# B&R Automation Studio project RS15_RX_30005_r00 (part 3)

#### A1_Basic.var - Local variables
```iecst
(********************************************************************
 * COPYRIGHT -- Microsoft
 ********************************************************************
 * Program: A1_Basic
 * File: A1_Basic.var
 * Author: pkiel
 * Created: July 11, 2011
 ********************************************************************
 * Local variables of program A1_Basic
 ********************************************************************)
VAR
	AutoAck : BOOL;
	AxisErrorNcAccess : UINT;
	DriveStatus : MC_DRIVESTATUS_TYP;
	HomeRestore : BOOL;
	InitEndlessPosition : BOOL;
	InitModPos_Done : BOOL;
	InitModPosition : BOOL;
  iiSetPosCount : DINT;
  iiSetPosCount1 : DINT;
  rSetPosCount1 : REAL;
  rMotorTemp : REAL;
  rAxisTimSet_SP_Vel  : REAL ; (*Set point Velocity for Axis manual timing setting cycle, in units/s*)
  rAxisTimSet_SP_Acc  : REAL ; (*Set point Acceleration for Axis manual timing setting cycle, in units/s²*)
  rAxisTimSet_SP_Dec  : REAL ; (*Set point Deceleration for Axis manual timing setting cycle, in units/s²*)
  uiAxisTimSet_SP_Dir : USINT ; (*Set point Direction for Axis manual timing setting cycle*)
  uiAxisTimSet_SP_ShiftAppMode : UINT ; (*Set point Shit Application mode for phasing Axis manual timing setting cycle*)
	MC_BR_InitEndlessPosition_0 : MC_BR_InitEndlessPosition;
	MC_BR_InitModPos_0 : MC_BR_InitModPos;
	MC_BR_Phasing_0 : MC_BR_Phasing;
	MC_BR_ReadDriveStatus_0 : MC_BR_ReadDriveStatus;
	MC_Home_0 : MC_Home;
	MC_Home_1 : MC_Home;
  MC_MoveVelocity_0 : MC_MoveVelocity;
  MC_MoveVelocity_1 : MC_MoveVelocity;
	MC_Power_0 : MC_Power;
	MC_ReadActualPosition_0 : MC_ReadActualPosition;
	MC_ReadActualTorque_0 : MC_ReadActualTorque;
	MC_ReadActualVelocity_0 : MC_ReadActualVelocity;
	MC_ReadAxisError_0 : MC_ReadAxisError;
	MC_ReadStatus_0 : MC_ReadStatus;
	MC_Reset_0 : MC_Reset;
  MC_Stop_0 : MC_Stop;
  MC_Stop_1 : MC_Stop;
  MC_SetOverride_0 : MC_SetOverride ;
	ResetError : BOOL;
  bTest_ : ARRAY[0..9] OF  BOOL;
  rTempActPhasDeg : REAL;
  rA9PosCorDeg : REAL;

  iiSP_SlPos_U  : DINT ; (*On Slave side, input set point position of the position controller ParID 428, in unit*)
  rSP_SlPos_Deg : REAL ; (*On Slave side, input set point position of the position controller ParID 428, in deg*)
  iiSP_MaPos_U  : DINT ; (*On Master side, input set point position of the position controller ParID 412, in unit*)
  rSP_MaPos_Deg : REAL ; (*On Master side, input set point position of the position controller ParID 412, in deg*)
  MC_BR_CyclicRead_0 : MC_BR_CyclicRead ;
  MC_BR_CyclicRead_1 : MC_BR_CyclicRead ;
  rTempPosA1_Deg : REAL;

  uiiMemoNumRev : UDINT ;
END_VAR
```

### Program Logical/BagMachine_Section/Perf/Axis1/A1_CamProfCalc

#### A1_CamProfCalc.var
```iecst
(********************************************************************
 * COPYRIGHT -- .
 ********************************************************************
 * Program: A1_CamProfCalc
 * File: A1_CamProfCalc.var
 * Author: dominique
 * Created: August 24, 2011
 ********************************************************************
 * Local variables of program A1_CamProfCalc
 ********************************************************************)

VAR
  stPerfCamSect : MC_CAM_SECTIONS_TYP ;
  stPerfCamProf : MC_CAMPROFILE_TYP ;
  MC_BR_CalcCamFromSections_0    : MC_BR_CalcCamFromSections ;
  MC_BR_DownloadCamProfileData_0 : MC_BR_DownloadCamProfileData ;
  MC_BR_GetCamMasterPosition_1   : MC_BR_GetCamMasterPosition ;
  MC_BR_GetCamMasterPosition_2   : MC_BR_GetCamMasterPosition ;
  MC_BR_GetCamSlavePosition_0    : MC_BR_GetCamSlavePosition ;
  MC_Home_0                      : MC_Home ;

  rMaInterval    : REAL ;
  rSlInterval    : REAL ;
  rSlPeriod      : REAL ;
  iiSlEndPoint   : DINT ;
  rSpeedInterval : REAL ;
  iStepCalPerfCam : INT ;
  bNextStep : BOOL ;
  bTestMode : BOOL ;

  iStepPosPerfCam : INT ;
  rCamMaPosition  : REAL ;
  rCamMaPos       : REAL ;
  rCamMaStartPos  : REAL ;
  rCamSlPosition  : REAL ;
  rCamSlPos       : REAL ;
  rCamSlPosCalc   : REAL ;
  rPosParkSlaveCamDeg   : REAL ;
  rTempPosParkSlaveCam  : REAL ;
  rTempPosParkMasterCam : REAL ;
  rMastMatchedSpeed : REAL ;
  bCmd_CalcCam_Test : BOOL ;
END_VAR

VAR CONSTANT

END_VAR
```

#### A1_CamProfCalcCyclic.st
```iecst
(********************************************************************
 * COPYRIGHT -- .
 ********************************************************************
 * Program: A1_CamProfCalc
 * File: A1_CamProfCalcCyclic.st
 * Author: dominique
 * Created: August 24, 2011
 ********************************************************************
 * Implementation of program A1_CamProfCalc
 ********************************************************************)

PROGRAM _CYCLIC

    IF ( gA[1].Cmd_CalcCameProf OR
         0                      OR
         bCmd_CalcCam_Test )    AND
       (iStepCalPerfCam = 0)    AND
       (iStepPosPerfCam = 0)    AND
       //0                        AND
       1                        THEN
      iStepCalPerfCam := 2 ;
    END_IF ;

    CASE iStepCalPerfCam OF

      // -------------------------------------------------------------------------------
      1 : ; // Waiting Error Reset
        IF EDGEPOS(gAlarmReset OR gA[1].Cmd_Reset) THEN
          g_bCamPerfCalcReset    := 0 ;
          g_bCamPerfCalc_Error   := 0 ;
          g_uiCalcCamPerfErrorID := 0 ;
          iStepCalPerfCam := 0 ;
        END_IF

      // -------------------------------------------------------------------------------
      2 : ; // Came profile calculation

        // Came profile calculation just for pos park on master side calculation
        // Synchro zone de 0° --> End Point of synchro zone
        // Compensation zone End Point of synchro zone --> Axis Periode

        // Calculation of Came section
        // Slave interval
        rSlInterval := gSP_A[1].MatchedSpeed * gA[1].UnitsPerDeg ;
        // Master interval
        rMaInterval := g_rActualSizePerf_in / gRecipeActive.Repeat * rSlInterval ;
        // Speed inteval
        rSpeedInterval := rSlInterval / rMaInterval ;
        // Slave Periode
        rSlPeriod := gA[1].AxisPeriod / gSP_PerfKnifeCount ;
        // Slave end point
        iiSlEndPoint := REAL_TO_DINT(rSlPeriod) ;
        // Master matched speed zone
        rMastMatchedSpeed := g_rActualSizePerf_in / gRecipeActive.Repeat * gSP_A[1].MatchedSpeed ;

        // First point of the Came Profile
        stPerfCamSect.Section[0].MasterPosition   := 0.0 ;
        stPerfCamSect.Section[0].SlavePosition    := 0.0 ;
        stPerfCamSect.Section[0].FirstDerivative  := rSpeedInterval ;
        stPerfCamSect.Section[0].SecondDerivative := 0.0 ;
        stPerfCamSect.Section[0].Mode             := mcABSOLUTE ;
        stPerfCamSect.Section[0].Type             := mcSTRAIGHT_LINE ;

        // Second point of the Came Profile
        stPerfCamSect.Section[1].MasterPosition   := rMaInterval ;
        stPerfCamSect.Section[1].SlavePosition    := rSlInterval ;
        stPerfCamSect.Section[1].FirstDerivative  := rSpeedInterval ;
        stPerfCamSect.Section[1].SecondDerivative := 0.0 ;
        stPerfCamSect.Section[1].Mode             := mcABSOLUTE ;
        stPerfCamSect.Section[1].Type             := mc5TH_ORDER_POLYNOMIAL ;

        // Third point of the Came Profile
        stPerfCamSect.Section[2].MasterPosition   := REAL_TO_DINT(gA[11].AxisPeriod) ;
        stPerfCamSect.Section[2].SlavePosition    := iiSlEndPoint ;
        stPerfCamSect.Section[2].FirstDerivative  := rSpeedInterval ;
        stPerfCamSect.Section[2].SecondDerivative := 0.0 ;
        stPerfCamSect.Section[2].Mode             := mcABSOLUTE ;
        stPerfCamSect.Section[2].Type             := mcLAST_POINT ;

        MC_BR_CalcCamFromSections_0.Execute           := 1 ;
        MC_BR_CalcCamFromSections_0.DataAddress       := ADR(stPerfCamSect) ;
        MC_BR_CalcCamFromSections_0.CamProfileAddress := ADR(stPerfCamProf) ;

        iStepCalPerfCam := 3 ;

      // -------------------------------------------------------------------------------
      3 : ; // Waiting result of the function
        IF MC_BR_CalcCamFromSections_0.Done AND
           ( bNextStep OR NOT(bTestMode) )  THEN
          MC_BR_CalcCamFromSections_0.Execute := 0 ;
          iStepCalPerfCam := 4 ;
          bNextStep := 0 ;
        ELSIF MC_BR_CalcCamFromSections_0.Error THEN
          g_uiCalcCamPerfErrorID := MC_BR_CalcCamFromSections_0.ErrorID;
          IF ( bNextStep OR NOT(bTestMode) ) THEN
            MC_BR_CalcCamFromSections_0.Execute :=0 ;
            g_bCamPerfCalc_Error := 1 ;
            bNextStep := 0 ;
            iStepCalPerfCam := 1 ;
          END_IF
        END_IF

      // -------------------------------------------------------------------------------
      4 : ; // Transfer Came to the Drive
        MC_BR_DownloadCamProfileData_0.Axis        := gA[1].Ident ;
        MC_BR_DownloadCamProfileData_0.DataAddress := ADR(stPerfCamProf) ;
        MC_BR_DownloadCamProfileData_0.Index       := g_uiIndexCamProfPerf ;
        MC_BR_DownloadCamProfileData_0.Periodic    := mcPERIODIC ;
        MC_BR_DownloadCamProfileData_0.Execute     := 1 ;

        iStepCalPerfCam := 5 ;

      // -------------------------------------------------------------------------------
      5 : ; // Waiting result of the function
        IF MC_BR_DownloadCamProfileData_0.Done AND
           ( bNextStep OR NOT(bTestMode) )     THEN
          MC_BR_DownloadCamProfileData_0.Execute:=FALSE;
          gA[1].Cmd_GetMaPosProf := 1 ;
          gA[1].Cmd_CalcCameProf := 0 ;
          bCmd_CalcCam_Test := 0 ;
          bNextStep := 0 ;
          iStepCalPerfCam := 0 ;
        ELSIF MC_BR_DownloadCamProfileData_0.Error THEN
          g_uiCalcCamPerfErrorID := MC_BR_DownloadCamProfileData_0.ErrorID;
          IF ( bNextStep OR NOT(bTestMode) ) THEN
            MC_BR_DownloadCamProfileData_0.Execute := 0 ;
            g_bCamPerfCalc_Error := 1 ;
            bNextStep := 0 ;
            iStepCalPerfCam := 1 ;
          END_IF
        END_IF
    END_CASE

    MC_BR_CalcCamFromSections_0() ;
    MC_BR_DownloadCamProfileData_0() ;

    // In Came Profile master position calculation according to the slave position
    IF ( gA[1].Cmd_GetMaPosProf   OR
         gA[1].Cmd_GetSlPosProf ) AND
       (iStepPosPerfCam = 0)      AND
       //0                          AND
       1                          THEN
      iStepPosPerfCam := 2 ;

      g_uiGetPosCamProfErrorID_1 := 0 ;
      g_uiGetPosCamProfErrorID_2 := 0 ;
      g_uiGetPosCamProfErrorID_3 := 0 ;
      g_uiHomCamProfErrorID      := 0 ;
    END_IF ;

    CASE iStepPosPerfCam OF
      // -------------------------------------------------------------------------------
      1 : ;// Waiting Error Reset
        IF EDGEPOS(gAlarmReset OR gA[1].Cmd_Reset) THEN
          iStepPosPerfCam := 0 ;
          g_bGetMaPosCamProfError_1 := 0 ;
          g_bGetMaPosCamProfError_2 := 0 ;
          g_bGetSlPosCamProfError   := 0 ;
          g_bHomeCamProfError       := 0 ;
        END_IF

      // -------------------------------------------------------------------------------
      2 : ; // Task selection
          IF gA[1].Cmd_GetMaPosProf THEN
            iStepPosPerfCam := 3 ;
          ELSIF gA[1].Cmd_GetSlPosProf THEN
            iStepPosPerfCam := 10 ;
          ELSE
            iStepPosPerfCam := 0 ;
          END_IF

      // -------------------------------------------------------------------------------
      3 : ; // Get Came master position command activation
        MC_BR_GetCamMasterPosition_1.Master := gA[11].Ident ;
        MC_BR_GetCamMasterPosition_1.Slave  := gA[1].Ident ;

        rCamSlPosCalc := H_FC_Modulus(IN_rMod:=rSlPeriod, IN_rVar:=gA[1].PositionCount) ;

        MC_BR_GetCamMasterPosition_1.Execute             := 1 ;
        MC_BR_GetCamMasterPosition_1.SlavePosition       := rCamSlPosCalc ;
        MC_BR_GetCamMasterPosition_1.MasterStartPosition := rCamMaStartPos ;
        MC_BR_GetCamMasterPosition_1.DataAddress         := ADR(stPerfCamProf) ;
        MC_BR_GetCamMasterPosition_1.MasterFactor        := 1 ;
        MC_BR_GetCamMasterPosition_1.SlaveFactor         := 1 ;
        IF MC_BR_GetCamMasterPosition_1.Done THEN
          rCamMaPosition := MC_BR_GetCamMasterPosition_1.MasterPosition ;
          MC_BR_GetCamMasterPosition_1.Execute := 0 ;
        ELSIF MC_BR_GetCamMasterPosition_1.Error THEN
          g_uiGetPosCamProfErrorID_1 := MC_BR_GetCamMasterPosition_1.ErrorID ;
          MC_BR_GetCamMasterPosition_1.Execute := 0 ;
          g_bGetMaPosCamProfError_1 := 1 ;
        END_IF

        MC_BR_GetCamMasterPosition_2.Master := gA[11].Ident ;
        MC_BR_GetCamMasterPosition_2.Slave  := gA[1].Ident ;

        rTempPosParkSlaveCam := gSP_A[1].ParkPosition * gA[1].UnitsPerDeg ;

        MC_BR_GetCamMasterPosition_2.Execute             := 1 ;
        MC_BR_GetCamMasterPosition_2.SlavePosition       := rTempPosParkSlaveCam ;
        MC_BR_GetCamMasterPosition_2.MasterStartPosition := rCamMaStartPos ;
        MC_BR_GetCamMasterPosition_2.DataAddress         := ADR(stPerfCamProf) ;
        MC_BR_GetCamMasterPosition_2.MasterFactor        := 1 ;
        MC_BR_GetCamMasterPosition_2.SlaveFactor         := 1 ;
        IF MC_BR_GetCamMasterPosition_2.Done AND
           NOT ( g_bGetMaPosCamProfError_1 ) THEN
          g_rPosParkMasterCam := MC_BR_GetCamMasterPosition_2.MasterPosition / gA[1].UnitsPerDeg ;
          MC_BR_GetCamMasterPosition_2.Execute := 0 ;
          iStepPosPerfCam := 4 ;
        ELSIF MC_BR_GetCamMasterPosition_2.Error THEN
          g_uiGetPosCamProfErrorID_2 := MC_BR_GetCamMasterPosition_2.ErrorID ;
          MC_BR_GetCamMasterPosition_2.Execute := 0 ;
          g_bGetMaPosCamProfError_2 := 1 ;
        END_IF

        IF g_bGetMaPosCamProfError_1 OR
           g_bGetMaPosCamProfError_2 THEN
          iStepPosPerfCam := 1 ;
        END_IF

      // -------------------------------------------------------------------------------
      4 : ; // Positionning Master on Synchro position
        MC_Home_0.Axis       := gA[11].Ident;
        IF gA[11].Ind_StandStill THEN
          MC_Home_0.Execute := 1 ;
        END_IF
        MC_Home_0.Position   := rCamMaPosition ;
        MC_Home_0.HomingMode := mcHOME_DIRECT;
        IF MC_Home_0.Done THEN
          MC_Home_0.Execute := 0 ;
          iStepPosPerfCam := 0 ;
          gA[1].Cmd_GetMaPosProf := 0 ;
          gA[1].Cmd_CalcCameProf := 0 ;
          g_bCameProf_OK := 1 ;
        ELSIF MC_Home_0.Error THEN
          g_uiHomCamProfErrorID := MC_Home_0.ErrorID ;
          MC_Home_0.Execute := 0 ;
          g_bHomeCamProfError := 1 ;
          iStepPosPerfCam := 1 ;
        END_IF

      // -------------------------------------------------------------------------------
      10 : ; // Get Came slave position command activation
        MC_BR_GetCamSlavePosition_0.Master := gA[11].Ident ;
        MC_BR_GetCamSlavePosition_0.Slave  := gA[1].Ident ;

        MC_BR_GetCamSlavePosition_0.Execute        := 1 ;
        MC_BR_GetCamSlavePosition_0.MasterPosition := rCamMaPos ;
        MC_BR_GetCamSlavePosition_0.DataAddress    := ADR(stPerfCamProf) ;
        MC_BR_GetCamSlavePosition_0.MasterFactor   := 1 ;
        MC_BR_GetCamSlavePosition_0.SlaveFactor    := 1 ;
        IF MC_BR_GetCamSlavePosition_0.Done THEN
          rCamSlPosition := MC_BR_GetCamSlavePosition_0.SlavePosition ;
          MC_BR_GetCamSlavePosition_0.Execute := 0 ;
          iStepPosPerfCam := 11 ;
        ELSIF MC_BR_GetCamSlavePosition_0.Error THEN
          g_uiGetPosCamProfErrorID_3 := MC_BR_GetCamSlavePosition_0.ErrorID ;
          MC_BR_GetCamSlavePosition_0.Execute := 0 ;
          g_bGetSlPosCamProfError := 1 ;
          iStepPosPerfCam := 1 ;
        END_IF

      // -------------------------------------------------------------------------------
      11 : ; //
        gA[1].Cmd_GetSlPosProf := 0 ;
        iStepPosPerfCam := 0 ;
      END_CASE

    MC_Home_0();
    MC_BR_GetCamMasterPosition_1() ;
    MC_BR_GetCamMasterPosition_2() ;
    MC_BR_GetCamSlavePosition_0() ;
END_PROGRAM
```

### Program Logical/BagMachine_Section/Perf/Axis1/A1_Control

#### A1_ControlCyclic.ld
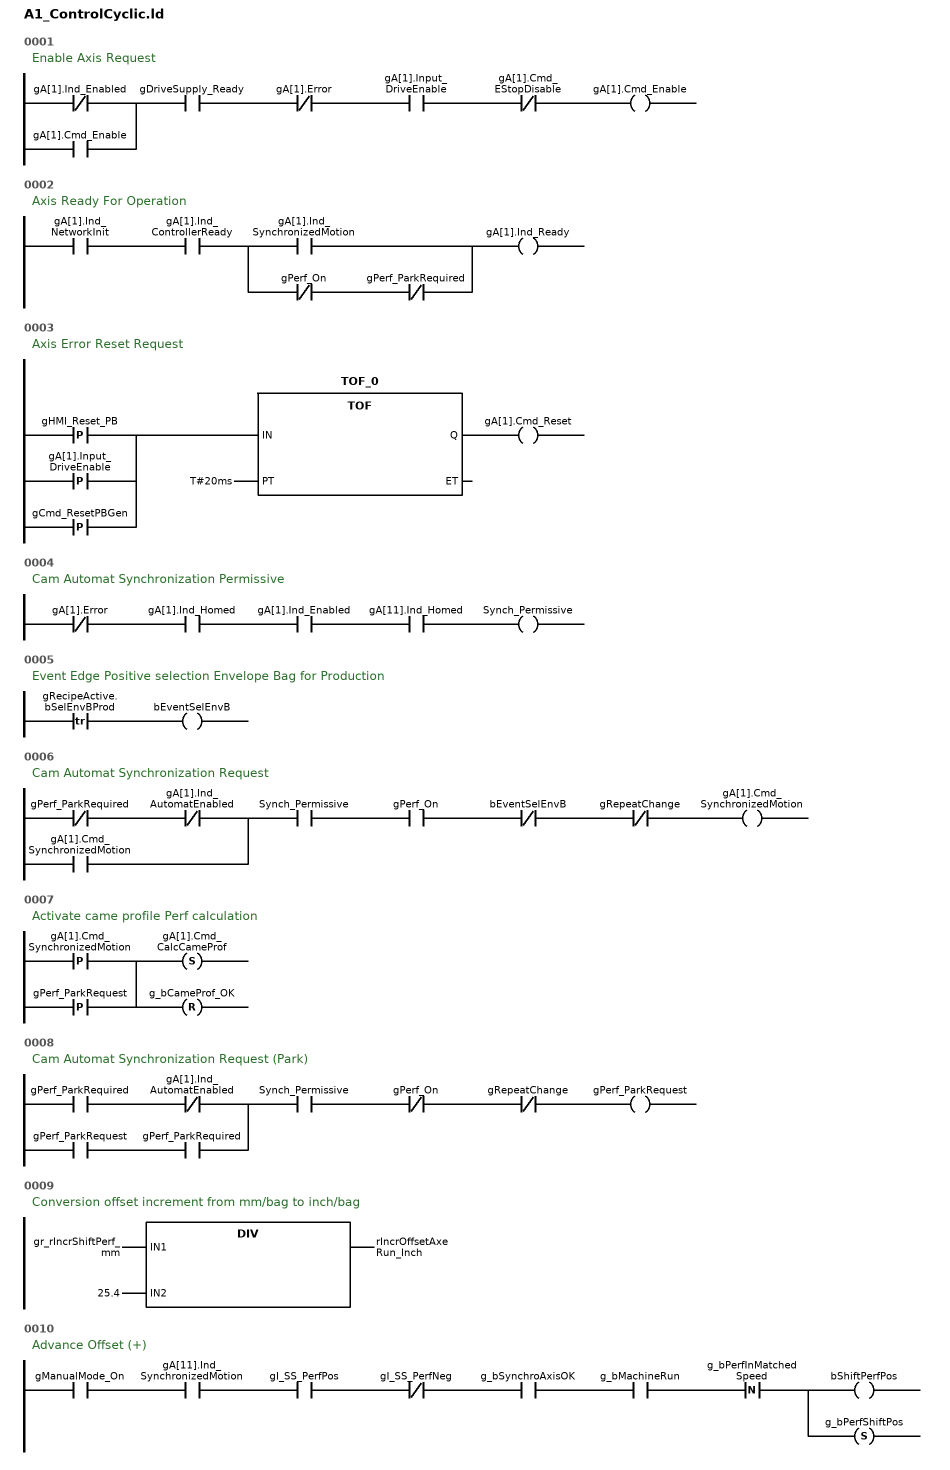
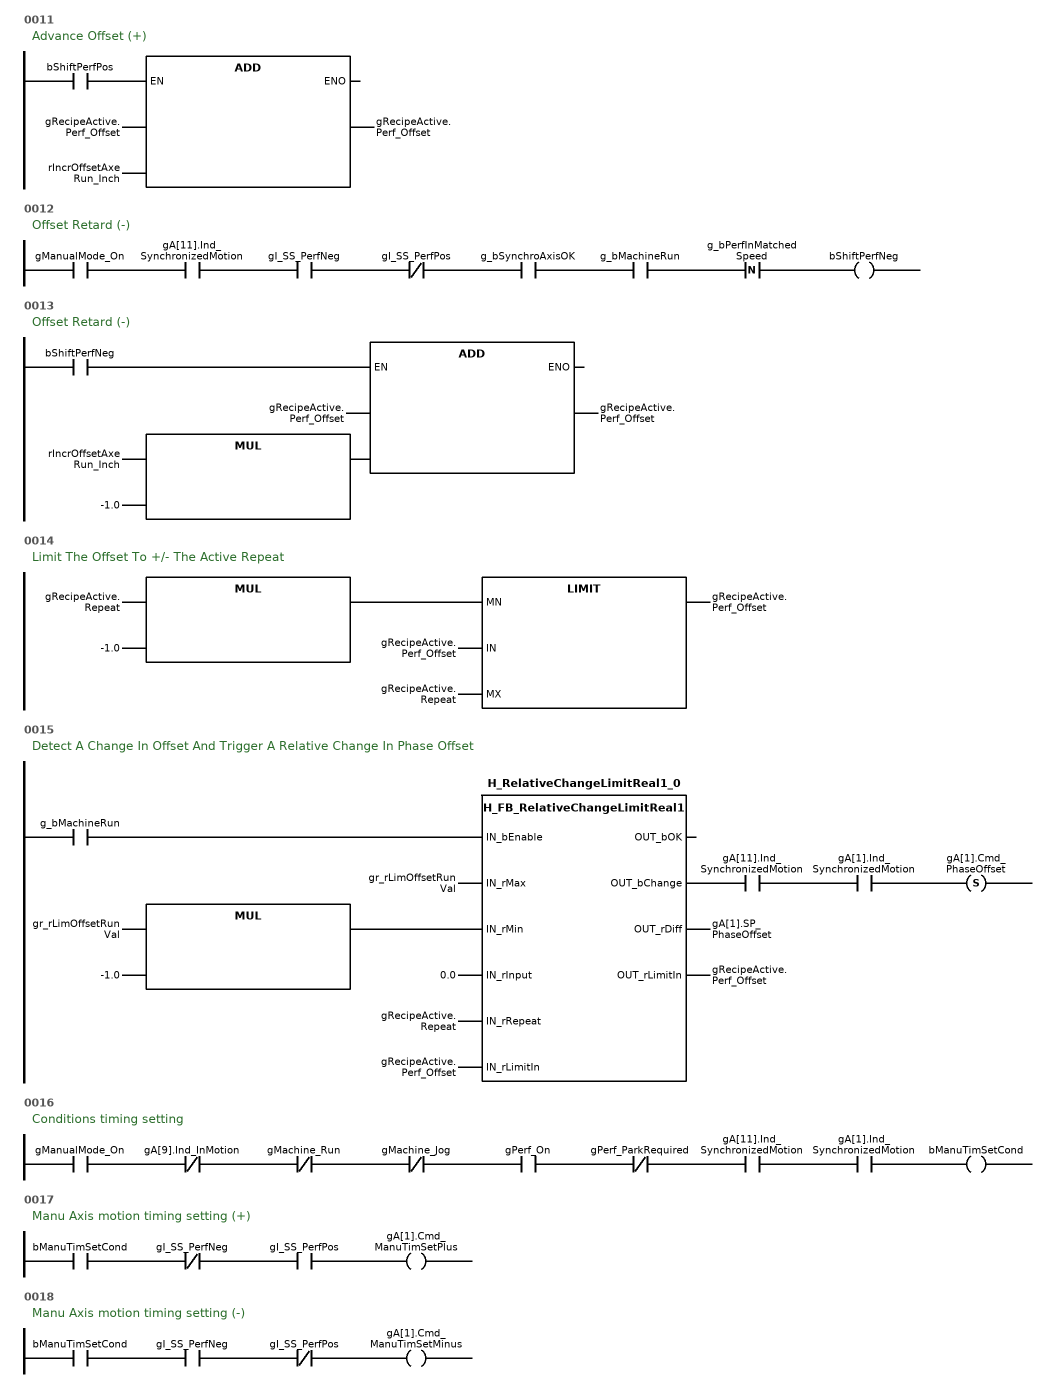
Ladder, written as Structured Text:
```iecst
(********************************************************************
 * COPYRIGHT -- Microsoft
 ********************************************************************
 * Program: A1_Control
 * File: A1_ControlCyclic.ld
 * Author: pkiel
 * Created: July 12, 2011
 ********************************************************************
 * Implementation of program A1_Control
 ********************************************************************)

PROGRAM _CYCLIC
VAR
    _p1 : BOOL;
    _e2 : R_TRIG;
    _e3 : R_TRIG;
    _e4 : R_TRIG;
    _e5 : R_TRIG;
    _e6 : R_TRIG;
    _e7 : F_TRIG;
    _p8 : BOOL;
    _e9 : F_TRIG;
END_VAR
(* Network 1: Enable Axis Request *)
gA[1].Cmd_Enable := (NOT gA[1].Ind_Enabled OR gA[1].Cmd_Enable) AND gDriveSupply_Ready AND NOT gA[1].Error AND gA[1].Input_DriveEnable AND NOT gA[1].Cmd_EStopDisable;

(* Network 2: Axis Ready For Operation *)
_p1 := gA[1].Ind_NetworkInit AND gA[1].Ind_ControllerReady;
gA[1].Ind_Ready := _p1 AND (gA[1].Ind_SynchronizedMotion OR (NOT gPerf_On AND NOT gPerf_ParkRequired));

(* Network 3: Axis Error Reset Request *)
_e2(CLK := gHMI_Reset_PB);
_e3(CLK := gA[1].Input_DriveEnable);
_e4(CLK := gCmd_ResetPBGen);
TOF_0(IN := _e2.Q OR _e3.Q OR _e4.Q, PT := T#20ms);
gA[1].Cmd_Reset := TOF_0.Q;

(* Network 4: Cam Automat Synchronization Permissive *)
Synch_Permissive := NOT gA[1].Error AND gA[1].Ind_Homed AND gA[1].Ind_Enabled AND gA[11].Ind_Homed;

(* Network 5: Event Edge Positive selection Envelope Bag for Production  *)
bEventSelEnvB := FALSE;

(* Network 6: Cam Automat Synchronization Request *)
gA[1].Cmd_SynchronizedMotion := ((NOT gPerf_ParkRequired AND NOT gA[1].Ind_AutomatEnabled) OR gA[1].Cmd_SynchronizedMotion) AND Synch_Permissive AND gPerf_On AND NOT bEventSelEnvB AND NOT gRepeatChange;

(* Network 7: Activate came profile Perf calculation  *)
_e5(CLK := gA[1].Cmd_SynchronizedMotion);
_e6(CLK := gPerf_ParkRequest);
IF _e5.Q OR _e6.Q THEN
    gA[1].Cmd_CalcCameProf := TRUE;
    g_bCameProf_OK := FALSE;
END_IF;

(* Network 8: Cam Automat Synchronization Request (Park) *)
gPerf_ParkRequest := ((gPerf_ParkRequired AND NOT gA[1].Ind_AutomatEnabled) OR (gPerf_ParkRequest AND gPerf_ParkRequired)) AND Synch_Permissive AND NOT gPerf_On AND NOT gRepeatChange;

(* Network 9: Conversion offset increment from mm/bag to inch/bag *)
rIncrOffsetAxeRun_Inch := gr_rIncrShiftPerf_mm / 25.4;

(* Network 10: Advance Offset (+) *)
_e7(CLK := g_bPerfInMatchedSpeed);
_p8 := gManualMode_On AND gA[11].Ind_SynchronizedMotion AND gI_SS_PerfPos AND NOT gI_SS_PerfNeg AND g_bSynchroAxisOK AND g_bMachineRun AND _e7.Q;
bShiftPerfPos := _p8;
IF _p8 THEN g_bPerfShiftPos := TRUE; END_IF;

(* Network 11: Advance Offset (+) *)
IF bShiftPerfPos THEN
    gRecipeActive.Perf_Offset := gRecipeActive.Perf_Offset + rIncrOffsetAxeRun_Inch;
END_IF;

(* Network 12: Offset Retard (-) *)
_e9(CLK := g_bPerfInMatchedSpeed);
bShiftPerfNeg := gManualMode_On AND gA[11].Ind_SynchronizedMotion AND gI_SS_PerfNeg AND NOT gI_SS_PerfPos AND g_bSynchroAxisOK AND g_bMachineRun AND _e9.Q;

(* Network 13: Offset Retard (-) *)
IF bShiftPerfNeg THEN
    gRecipeActive.Perf_Offset := gRecipeActive.Perf_Offset + (rIncrOffsetAxeRun_Inch * -1.0);
END_IF;

(* Network 14: Limit The Offset To +/- The Active Repeat *)
gRecipeActive.Perf_Offset := LIMIT(MN := gRecipeActive.Repeat * -1.0, IN := gRecipeActive.Perf_Offset, MX := gRecipeActive.Repeat);

(* Network 15: Detect A Change In Offset And Trigger A Relative Change In Phase Offset *)
H_RelativeChangeLimitReal1_0(IN_bEnable := g_bMachineRun, IN_rMax := gr_rLimOffsetRunVal, IN_rMin := gr_rLimOffsetRunVal * -1.0, IN_rInput := 0.0, IN_rRepeat := gRecipeActive.Repeat, IN_rLimitIn := gRecipeActive.Perf_Offset);
IF H_RelativeChangeLimitReal1_0.OUT_bChange AND gA[11].Ind_SynchronizedMotion AND gA[1].Ind_SynchronizedMotion THEN
    gA[1].Cmd_PhaseOffset := TRUE;
END_IF;
gA[1].SP_PhaseOffset := H_RelativeChangeLimitReal1_0.OUT_rDiff;
gRecipeActive.Perf_Offset := H_RelativeChangeLimitReal1_0.OUT_rLimitIn;

(* Network 16: Conditions timing setting  *)
bManuTimSetCond := gManualMode_On AND NOT gA[9].Ind_InMotion AND NOT gMachine_Run AND NOT gMachine_Jog AND gPerf_On AND NOT gPerf_ParkRequired AND gA[11].Ind_SynchronizedMotion AND gA[1].Ind_SynchronizedMotion;

(* Network 17: Manu Axis motion timing setting (+) *)
gA[1].Cmd_ManuTimSetPlus := bManuTimSetCond AND NOT gI_SS_PerfNeg AND gI_SS_PerfPos;

(* Network 18: Manu Axis motion timing setting (-) *)
gA[1].Cmd_ManuTimSetMinus := bManuTimSetCond AND gI_SS_PerfNeg AND NOT gI_SS_PerfPos;
END_PROGRAM
```

### Program Logical/BagMachine_Section/Perf/Axis1/A1_Cycle (IEC)

#### A1_CycleInit.st - Initialization code
```iecst
(********************************************************************
 * COPYRIGHT -- .
 ********************************************************************
 * Program: A1_Cycle
 * File: A1_CycleInit.st
 * Author: dominique
 * Created: August 01, 2011
 ********************************************************************
 * Implementation of program A1_Cycle
 ********************************************************************)

PROGRAM _INIT

(* TODO : Add your code here *)

END_PROGRAM
```

### A1_Init.ax
```
InitParameter (Version=2.24.0, NcSwId=ACP10)
  ACP10AXIS_typ:
    dig_in:
      level:
        reference = ncACTIV_HI
        pos_hw_end = ncACTIV_HI
        neg_hw_end = ncACTIV_HI
        trigger1 = ncACTIV_HI
        trigger2 = ncACTIV_HI
    encoder_if:
      parameter:
        count_dir = ncSTANDARD
        scaling:
          load:
            units = 18000
            rev_motor = 1
    limit:
      parameter:
        v_pos = 1.8e+006
        v_neg = 1.8e+006
        a1_pos = 5e+006
        a2_pos = 5e+006
        a1_neg = 5e+006
        a2_neg = 5e+006
        t_jolt = 0.0
        t_in_pos = 0.0
        pos_sw_end = 8388607
        neg_sw_end = -8388608
        ds_warning = 500.0
        ds_stop = 1000.0
        a_stop = 1e+030
        dv_stop = 0
        dv_stop_mode = ncOFF
    controller:
      mode = ncPOSITION
      position:
        kv = 400.0
        tn = 0.0
        t_predict = 0.0004
        t_total = 0.0012
        p_max = 1e+030
        i_max = 0.0
      speed:
        kv = 20.0
        tn = 0.0
        t_filter = 0.0
        isq_filter1:
          type = ncNOTCH
          a0 = 1321.0
          a1 = 400.0
          b0 = 0.0
          b1 = 0.0
          b2 = 0.0
          c0_par_id = 0
          c1_par_id = 0
        isq_filter2:
          type = ncOFF
          a0 = 0.0
          a1 = 0.0
          b0 = 0.0
          b1 = 0.0
          b2 = 0.0
          c0_par_id = 0
          c1_par_id = 0
        isq_filter3:
          type = ncOFF
          a0 = 0.0
          a1 = 0.0
          b0 = 0.0
          b1 = 0.0
          b2 = 0.0
          c0_par_id = 0
          c1_par_id = 0
      uf:
        type = ncLINEAR
        auto_config = ncMOTOR_PAR
        u0 = 0.0
        un = 0.0
        fn = 50.0
        k_f_slip = 0.0
      ff:
        torque_load = 0.0
        torque_pos = 0.0
        torque_neg = 0.0
        kv_torque = 0.0
        inertia = 0.0
        t_filter_a = 0.0
    move:
      stop:
        parameter[0]:
          decel_ramp = ncA_LIMIT
          controller = ncON
        parameter[1]:
          decel_ramp = ncA_LIMIT
          controller = ncON
        parameter[2]:
          decel_ramp = ncA_LIMIT
          controller = ncON
        parameter[3]:
          decel_ramp = ncA_LIMIT
          controller = ncON
        quickstop:
          decel_ramp = ncA_LIMIT
        drive_error:
          decel_ramp = ncA_LIMIT
      homing:
        parameter:
          s = 0
          v_switch = 5000.0
          v_trigger = 500.0
          a = 50000.0
          mode = ncHOME_OFFSET
          edge_sw = ncPOSITIVE
          start_dir = ncPOSITIVE
          trigg_dir = ncPOSITIVE
          ref_pulse = ncOFF
          tr_s_block = 0.0
      basis:
        parameter:
          v_pos = 36000.0
          v_neg = 100000.0
          a1_pos = 50000.0
          a2_pos = 50000.0
          a1_neg = 50000.0
          a2_neg = 50000.0
    message:
      text:
        parameter:
          format = ncBREAK
          columns = 80
          data_modul = Error_Eng
```

- Data object Logical/BagMachine_Section/Perf/Axis1/A1_Par (Apt) (no source held here)

### Program Logical/BagMachine_Section/Perf/Axis1/A1_Ref

#### A1_RefCyclic.ld
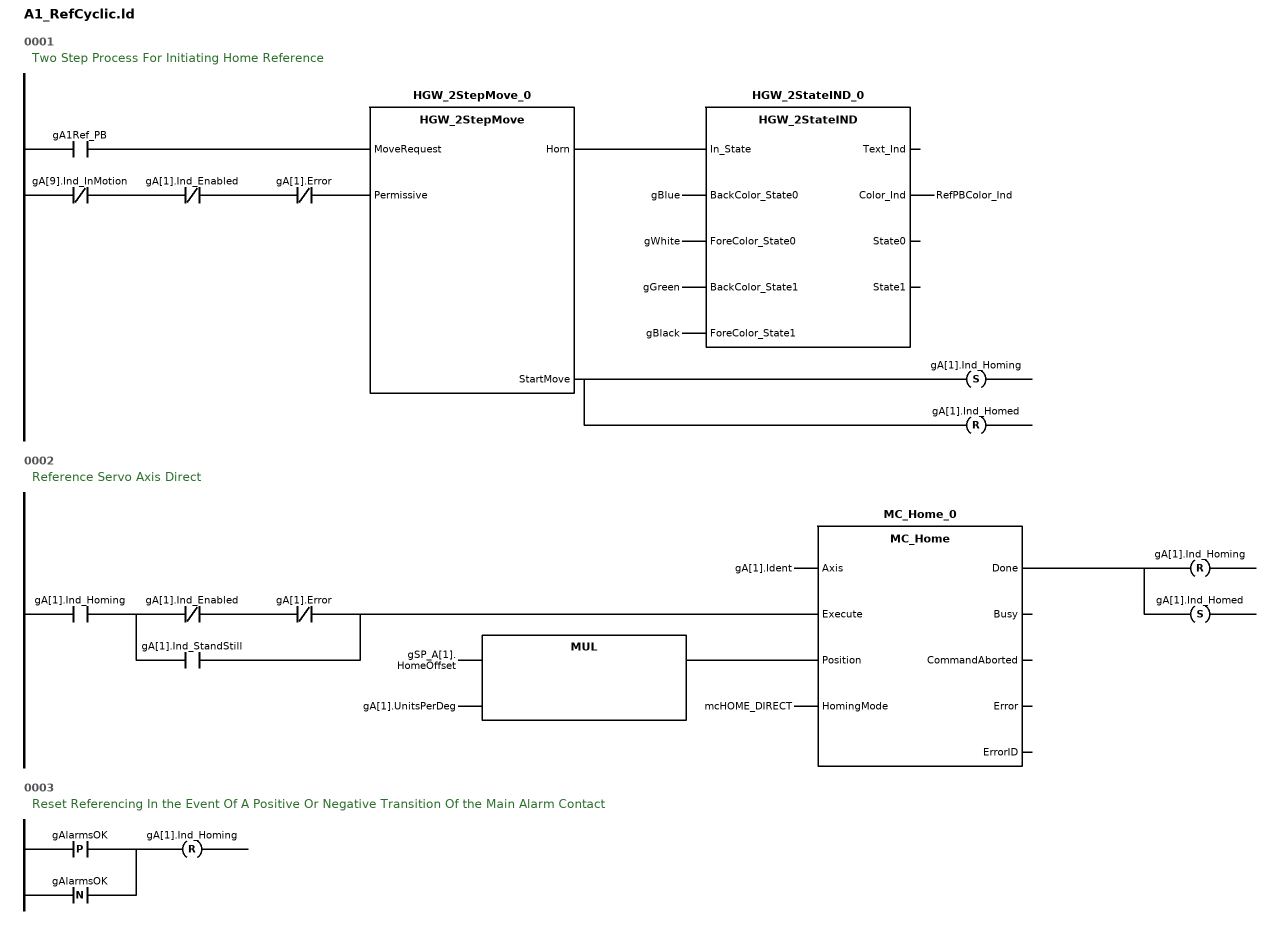
Ladder, written as Structured Text:
```iecst
(********************************************************************
 * COPYRIGHT -- Microsoft
 ********************************************************************
 * Program: A1_Ref
 * File: A1_RefCyclic.ld
 * Author: pkiel
 * Created: July 13, 2011
 ********************************************************************
 * Implementation of program A1_Ref
 ********************************************************************)

PROGRAM _CYCLIC
VAR
    _e1 : R_TRIG;
    _e2 : F_TRIG;
END_VAR
(* Network 1: Two Step Process For Initiating Home Reference *)
HGW_2StepMove_0(MoveRequest := gA1Ref_PB, Permissive := NOT gA[9].Ind_InMotion AND NOT gA[1].Ind_Enabled AND NOT gA[1].Error);
HGW_2StateIND_0(In_State := HGW_2StepMove_0.Horn, BackColor_State0 := gBlue, ForeColor_State0 := gWhite, BackColor_State1 := gGreen, ForeColor_State1 := gBlack);
RefPBColor_Ind := HGW_2StateIND_0.Color_Ind;
IF HGW_2StepMove_0.StartMove THEN
    gA[1].Ind_Homing := TRUE;
    gA[1].Ind_Homed := FALSE;
END_IF;

(* Network 2: Reference Servo Axis Direct *)
MC_Home_0(Axis := gA[1].Ident, Execute := gA[1].Ind_Homing AND ((NOT gA[1].Ind_Enabled AND NOT gA[1].Error) OR gA[1].Ind_StandStill), Position := gSP_A[1].HomeOffset * gA[1].UnitsPerDeg, HomingMode := mcHOME_DIRECT);
IF MC_Home_0.Done THEN
    gA[1].Ind_Homing := FALSE;
    gA[1].Ind_Homed := TRUE;
END_IF;

(* Network 3: Reset Referencing In the Event Of A Positive Or Negative Transition Of the Main Alarm Contact *)
_e1(CLK := gAlarmsOK);
_e2(CLK := gAlarmsOK);
IF _e1.Q OR _e2.Q THEN gA[1].Ind_Homing := FALSE; END_IF;
END_PROGRAM
```

- Data object Logical/BagMachine_Section/Perf/Axis11_VirtualAxis/A11_Init (Vax) - Virtual Axis Initialization File (no source held here)

- Data object Logical/BagMachine_Section/Perf/Axis11_VirtualAxis/A11_Par (Apt) - Virtual Axis Parameter File (no source held here)

### Program Logical/BagMachine_Section/Perf/Axis11_VirtualAxis/A11_Basic (IEC) - Basic Servo

#### A11_Basic.var
```iecst
(********************************************************************
 * COPYRIGHT -- Microsoft
 ********************************************************************
 * Program: A11_Basic
 * File: A11_Basic.var
 * Author: pkiel
 * Created: July 22, 2011
 ********************************************************************
 * Local variables of program A11_Basic
 ********************************************************************)
VAR
	AutoAck : BOOL;
	AxisErrorNcAccess : UINT;
	DriveStatus : MC_DRIVESTATUS_TYP;
	ErrorID : UINT;
	HomeRestore : BOOL;
	InitEndlessPosition : BOOL;
	InitModPos_Done : BOOL;
	InitModPosition : BOOL;
	MC_BR_InitEndlessPosition_0 : MC_BR_InitEndlessPosition;
	MC_BR_InitModPos_0 : MC_BR_InitModPos;
	MC_BR_Phasing_0 : MC_BR_Phasing;
  MC_BR_Phasing_1 : MC_BR_Phasing;
	MC_BR_ReadDriveStatus_0 : MC_BR_ReadDriveStatus;
	MC_Home_0 : MC_Home;
	MC_Home_1 : MC_Home;
	MC_MoveVelocity_0 : MC_MoveVelocity;
	MC_ReadActualPosition_0 : MC_ReadActualPosition;
	MC_ReadActualVelocity_0 : MC_ReadActualVelocity;
	MC_ReadAxisError_0 : MC_ReadAxisError;
	MC_ReadStatus_0 : MC_ReadStatus;
	MC_Reset_0 : MC_Reset;
	MC_Stop_0 : MC_Stop;
  stTON_O : TON ;
	ResetError : BOOL;
  rTemp_ : ARRAY[0..9] OF REAL ;
  bTest_ : ARRAY[0..9] OF BOOL ;
  rTest_ : ARRAY[0..9] OF REAL ;
  rAxisTimSet_SP_Vel  : REAL ; (*Set point Velocity for Axis manual timing setting cycle, in units/s*)
  rAxisTimSet_SP_Acc  : REAL ; (*Set point Acceleration for Axis manual timing setting cycle, in units/s²*)
  rAxisTimSet_SP_Dec  : REAL ; (*Set point Deceleration for Axis manual timing setting cycle, in units/s²*)
  uiAxisTimSet_SP_Dir : USINT ; (*Set point Direction for Axis manual timing setting cycle*)
  uiAxisTimSet_SP_ShiftAppMode : UINT ; (*Set point Shit Application mode for phasing Axis manual timing setting cycle*)
  rTempActPhasDeg : REAL;
  rA9PosCorDeg : REAL;
  MC_SetOverride_0 : MC_SetOverride;

  iiSP_SlPos_U  : DINT ; (*On Slave side, input set point position of the position controller ParID 428, in unit*)
  rSP_SlPos_Deg : REAL ; (*On Slave side, input set point position of the position controller ParID 428, in deg*)
  iiSP_MaPos_U  : DINT ; (*On Master side, input set point position of the position controller ParID 412, in unit*)
  rSP_MaPos_Deg : REAL ; (*On Master side, input set point position of the position controller ParID 412, in deg*)
  MC_BR_CyclicRead_0 : MC_BR_CyclicRead ;
  MC_BR_CyclicRead_1 : MC_BR_CyclicRead ;
  iIndex : INT;
  st_TON_0 : TON;
END_VAR
```

#### A11_BasicCyclic.st
```iecst
(********************************************************************
 * COPYRIGHT -- Microsoft
 ********************************************************************
 * Program: A11_Basic
 * File: A11_BasicCyclic.st
 * Author: pkiel
 * Created: July 22, 2011
 ********************************************************************
 * Implementation of program A11_Basic
 ********************************************************************)

PROGRAM _CYCLIC

	gA[11].UnitsPerInch := gA[11].AxisPeriod/gRecipeActive.Repeat;
  gA[11].InchPerDeg := gRecipeActive.Repeat / 360 ;

	IF (gA[11].Ident<>0) THEN

	(************************ READ DRIVE STATUS *************************)
	(* Access to the following bools:
	gA[x]_DriveStatus.Simulation			: If TRUE, simulation mode is active
	gA[x]_DriveStatus.NetworkInit			: If TRUE, the network is initialized
	gA[x]_DriveStatus.HomeSwitch			: If TRUE, the digital reference switch input is active
	gA[x]_DriveStatus.PosHWSwitch			: If TRUE, the positive hardware end switch is active
	gA[x]_DriveStatus.NegHWSwitch			: If TRUE, the negative hardware end switch is active
	gA[x]_DriveStatus.Trigger1				: If TRUE, the first trigger input is active
	gA[x]_DriveStatus.Trigger2				: If TRUE, the second trigger input is active
	gA[x]_DriveStatus.DriveEnable			: If TRUE, the enable input is active
	gA[x]_DriveStatus.ControllerReady		: If TRUE, the controller is ready to beturned on
	gA[x]_DriveStatus.ControllerStatus		: If TRUE, the controller is turned on (Same as MC_Power.Status)
	gA[x]_DriveStatus.AxisError				: If TRUE, at least one error has occurred (not acknowledged)
	gA[x]_DriveStatus.LagWarning			: If TRUE, the lag error has exceeded the limit value specified for a warning*)
		MC_BR_ReadDriveStatus_0.Enable := 1;
		MC_BR_ReadDriveStatus_0.Axis := gA[11].Ident;
		MC_BR_ReadDriveStatus_0.AdrDriveStatus := ADR (DriveStatus);
		MC_BR_ReadDriveStatus_0();
		gA[11].Ind_Simulation		:=	DriveStatus.Simulation;
		gA[11].Ind_NetworkInit		:=	DriveStatus.NetworkInit;
		gA[11].Input_Home			:=	DriveStatus.HomeSwitch;
		gA[11].Input_PosHW			:=	DriveStatus.PosHWSwitch;
		gA[11].Input_NegHW			:=	DriveStatus.NegHWSwitch;
		gA[11].Input_Trigger1		:=	DriveStatus.Trigger1;
		gA[11].Input_Trigger2		:=	DriveStatus.Trigger2;
		gA[11].Input_DriveEnable		:=	DriveStatus.DriveEnable;
		gA[11].Ind_ControllerReady	:=	DriveStatus.ControllerReady;
		gA[11].Ind_ControllerStatus	:=	DriveStatus.ControllerStatus;
		gA[11].Error					:=	DriveStatus.AxisError;
		gA[11].Ind_LagWarning		:=	DriveStatus.LagWarning;

	(************************ READ AXIS ERROR **********************)
		MC_ReadAxisError_0.Enable := gA[11].Ind_NetworkInit;
		MC_ReadAxisError_0.Axis := gA[11].Ident;
		MC_ReadAxisError_0.DataAddress := ADR(gA[11].ErrorText);
		MC_ReadAxisError_0.DataLength := SIZEOF(gA[11].ErrorText);
		MC_ReadAxisError_0.DataObjectName := 'Error_Eng';
		MC_ReadAxisError_0();
		IF(MC_ReadAxisError_0.Valid) THEN
			gA[11].ErrorID := MC_ReadAxisError_0.AxisErrorID;
			gA[11].ErrorCount := MC_ReadAxisError_0.AxisErrorCount;
		END_IF
	(* Auto Acknowledge Errors *)
		IF (gA[11].Cmd_Reset AND (gA[11].ErrorCount<>0) AND NOT AutoAck) THEN
			AutoAck:=1;
		ELSE
			AutoAck:=0;
		END_IF
	(*Axis Error Acknowledge*)
		IF (EDGEPOS(AutoAck) OR EDGEPOS(gA[11].ErrorAck)) THEN
			MC_ReadAxisError_0.Acknowledge := 1;
		ELSE;
			MC_ReadAxisError_0.Acknowledge :=0;
		END_IF

	(************************ RESET AXIS ERROR **********************)
		IF (gA[11].Cmd_Reset AND (gA[11].ErrorCount=0) AND gA[11].ErrorStop) THEN
			MC_Reset_0.Execute:=1;
		END_IF
		IF (MC_Reset_0.Done) THEN
			MC_Reset_0.Execute:=0;
			gA[11].Cmd_Reset:=0;
			ResetError := 0;
		END_IF
		IF (MC_Reset_0.Error) THEN
			MC_Reset_0.Execute:=0;
			gA[11].Cmd_Reset:=0;
			ResetError := 1;
		END_IF
		MC_Reset_0.Axis:=gA[11].Ident;
		MC_Reset_0();

	(************************ READ AXIS STATUS *************************)
		MC_ReadStatus_0.Enable := gA[11].Ind_NetworkInit;
		MC_ReadStatus_0.Axis := gA[11].Ident;
		MC_ReadStatus_0();
		IF(MC_ReadStatus_0.Valid = TRUE)THEN
			gA[11].Ind_Enabled 			:= NOT (MC_ReadStatus_0.Disabled);
			gA[11].Ind_StandStill		:= MC_ReadStatus_0.StandStill;
			gA[11].Ind_Stopping			:= MC_ReadStatus_0.Stopping;
			gA[11].Ind_DiscreteMotion	:= MC_ReadStatus_0.DiscreteMotion;
			gA[11].Ind_ContinuousMotion	:= MC_ReadStatus_0.ContinuousMotion;
			gA[11].Ind_SynchronizedMotion:= MC_ReadStatus_0.SynchronizedMotion;
			gA[11].ErrorStop				:= MC_ReadStatus_0.Errorstop;
		END_IF

	(******************** INIT POSITION MODULUS  *********************)
		MC_BR_InitModPos_0.Execute:= InitModPosition;
		MC_BR_InitModPos_0.Axis:= gA[11].Ident;
		MC_BR_InitModPos_0.Period:= REAL_TO_UDINT(gA[11].AxisPeriod);
		MC_BR_InitModPos_0.Factor:=1;
		InitModPos_Done:=MC_BR_InitModPos_0.Done;
		MC_BR_InitModPos_0();

	(******************** INIT ENDLESS POSITION *********************)
		MC_BR_InitEndlessPosition_0.Execute:= InitModPos_Done;
		MC_BR_InitEndlessPosition_0.Axis:= gA[11].Ident;
		MC_BR_InitEndlessPosition_0.DataAddress:= ADR(gEndPosData[11]);
		IF (MC_BR_InitEndlessPosition_0.Done) THEN
			InitModPosition:=0;
			InitEndlessPosition:=0;
			HomeRestore:=1;
		END_IF
		MC_BR_InitEndlessPosition_0();

	(************************ HOME AXIS FIRST POWER UP **********************)
		IF (HomeRestore AND NOT gA11_FirstHomed) THEN
			MC_Home_0.Execute:=1;
		END_IF
		MC_Home_0.Axis:=gA[11].Ident;
		MC_Home_0.Position:=0;
		MC_Home_0.HomingMode:=mcHOME_DIRECT;
		IF (MC_Home_0.Done) THEN
			MC_Home_0.Execute:=0;
			gA11_FirstHomed:=1;
		END_IF
		MC_Home_0();

	(************************ HOME AXIS **********************)
		IF (gA11_FirstHomed)     AND
       //NOT(gA[11].Ind_Homed) AND
       //g_bPerfInMatchedSpeed AND
       //gA[1].Ind_Homed       AND
       1                     THEN
			MC_Home_1.Execute:=HomeRestore;
		END_IF
		MC_Home_1.Axis:=gA[11].Ident;
		MC_Home_1.Position:=0;
		MC_Home_1.HomingMode:=mcHOME_RESTORE_POS;
		IF (MC_Home_1.Done) THEN
			gA[11].Ind_Homed:=1;
			HomeRestore:=0;
		END_IF
		MC_Home_1();

	(******************** READ ACTUAL POSITION *********************)
		MC_ReadActualPosition_0.Enable:= gA[11].Ind_NetworkInit;
		MC_ReadActualPosition_0.Axis:= gA[11].Ident;
		MC_ReadActualPosition_0();
		IF(MC_ReadActualPosition_0.Valid = TRUE)THEN
			gA[11].PositionCount := MC_ReadActualPosition_0.Position;
			gA[11].PositionInch := gA[11].PositionCount/gA[11].UnitsPerInch;
			gA[11].PositionDeg := gA[11].PositionCount/gA[11].UnitsPerDeg;
		END_IF

  //******************** READ SET POINT POSITION *********************
    // Slave side  : ParID 412 S_SET_VAX1 : 412: VAX: Position
    // Master side : ParID 412 S_SET_VAX1 : 412: VAX: Position

    // Slave side
    MC_BR_CyclicRead_0.Axis        := gA[11].Ident ;
    MC_BR_CyclicRead_0.Enable      := gA[11].Ind_NetworkInit;
    MC_BR_CyclicRead_0.ParID       := 412 ;
    MC_BR_CyclicRead_0.DataAddress := ADR(iiSP_SlPos_U);
    MC_BR_CyclicRead_0.DataType    := ncPAR_TYP_DINT ;
    // Master side
    MC_BR_CyclicRead_1.Axis        := gA[9].Ident ;
    MC_BR_CyclicRead_1.Enable      := gA[11].Ind_NetworkInit;
    MC_BR_CyclicRead_1.ParID       := 412 ;
    MC_BR_CyclicRead_1.DataAddress := ADR(iiSP_MaPos_U);
    MC_BR_CyclicRead_1.DataType    := ncPAR_TYP_DINT ;

    IF MC_BR_CyclicRead_0.Valid THEN
      rSP_SlPos_Deg := iiSP_SlPos_U/gA[11].UnitsPerDeg ;
    ELSIF MC_BR_CyclicRead_0.Error THEN
      MC_BR_CyclicRead_0.Enable := 0 ;
    END_IF
    IF MC_BR_CyclicRead_1.Valid THEN
      rSP_MaPos_Deg := iiSP_MaPos_U/gA[9].UnitsPerDeg ;
    ELSIF MC_BR_CyclicRead_1.Error THEN
      MC_BR_CyclicRead_1.Enable := 0 ;
    END_IF
    MC_BR_CyclicRead_0();
    MC_BR_CyclicRead_1();

  //******************** READ ACTUAL OFFSET *********************
  IF gA[11].rRSynDen > 0.0 THEN
    rTempActPhasDeg := rSP_SlPos_Deg - gA[11].rRSynNum / gA[11].rRSynDen * rSP_MaPos_Deg ;
    gA[11].rActPhasDeg := H_FC_Modulus (
                              IN_rMod := 360 * gA[11].rRSynNum / gA[11].rRSynDen ,
                              IN_rVar := rTempActPhasDeg
                                      ) ;
  END_IF

	(******************** READ ACTUAL VELOCITY *********************)
		IF(MC_ReadActualVelocity_0.Error=TRUE) THEN
			MC_ReadActualVelocity_0.Enable:= 0;
		ELSE
			MC_ReadActualVelocity_0.Enable:= 1;
		END_IF
		MC_ReadActualVelocity_0.Axis:= gA[11].Ident;
		MC_ReadActualVelocity_0();
		IF(MC_ReadActualVelocity_0.Valid = TRUE)THEN
			gA[11].ActualVelocity := MC_ReadActualVelocity_0.Velocity*60/gA[11].SP_MotorPPR;
			IF (gA[11].ActualVelocity>1) THEN
				gA[11].Ind_InMotion:=1;
			ELSE
				gA[11].Ind_InMotion:=0;
			END_IF
		END_IF

	(************************ AXIS VELOCITY MOVE **********************)
		MC_MoveVelocity_0.Axis:=gA[11].Ident;
		MC_MoveVelocity_0.Velocity:=gA[11].SP_Velocity*gA[11].AxisPeriod/60;
		MC_MoveVelocity_0.Acceleration:=gA[11].SP_Accel;
		MC_MoveVelocity_0.Deceleration:=gA[11].SP_Decel;
		MC_MoveVelocity_0.Direction:=mcPOSITIVE_DIR;
		IF ((EDGEPOS(gA[11].Cmd_ContinuousMotion)) OR (EDGEPOS(gA[11].Cmd_ContinuousMotionUpdate))) THEN
			MC_MoveVelocity_0.Execute:=1;
		ELSE
			MC_MoveVelocity_0.Execute:=0;
		END_IF;
		MC_MoveVelocity_0();

  //************************ AXIS OVERRIDE **********************
    MC_SetOverride_0.Axis      := gA[11].Ident ;
    MC_SetOverride_0.Enable    := gA[11].Cmd_Override ;
    MC_SetOverride_0.VelFactor := gA[11].rSP_OverrideV ;
    MC_SetOverride_0.AccFactor := gA[11].rSP_OverrideA ;
    IF (MC_SetOverride_0.Enabled) OR
       (MC_SetOverride_0.Error)   THEN
      gA[11].Cmd_Override := 0 ;
    END_IF
    MC_SetOverride_0();

	(************************ AXIS STOP **********************)
		MC_Stop_0.Axis:=gA[11].Ident;
		IF (gA[11].Ind_ContinuousMotion AND NOT gA[11].Cmd_ContinuousMotion) THEN
			MC_Stop_0.Deceleration:=gA[11].SP_Decel;
			MC_Stop_0.Execute:=1;
		END_IF
		IF (MC_Stop_0.Done OR MC_Stop_0.CommandAborted OR MC_Stop_0.Error) THEN
			MC_Stop_0.Execute:=0;
		END_IF
		MC_Stop_0();

    (************************ SHIFTING PERF CONTROL **********************)
    IF (g_iMachType = C_iRS26) THEN
      g_iNumBagPerfTear := REAL_TO_INT(gr_rDistPerfTearRS26_mm/gRecipeActive.Repeat/25.4) ;
      IF gA[12].bInMach THEN // Case Enveloppe Bag
        IF gRecipeActive.bSelEnvBProd THEN // Case Enveloppe Bag On
          g_iNumBagPerfTear := REAL_TO_INT(gr_rDistPerfTearEnvBOn_mm/gRecipeActive.Repeat/25.4) ;
        ELSE
          IF (g_rNumbPliers=2) THEN  // Case Enveloppe Bag Off and bags size 2 grippers
            g_iNumBagPerfTear := REAL_TO_INT(gr_rDistPerfTearEnvBOff2_mm/gRecipeActive.Repeat/25.4) ;
          ELSE                       // Case Enveloppe Bag Off and bags size 4 grippers
            g_iNumBagPerfTear := REAL_TO_INT(gr_rDistPerfTearEnvBOff4_mm/gRecipeActive.Repeat/25.4) ;
          END_IF
        END_IF
      END_IF
    ELSIF (g_iMachType = C_iRS15) THEN
      g_iNumBagPerfTear := REAL_TO_INT(gr_rDistPerfTearRS15_mm/gRecipeActive.Repeat/25.4) ;
    END_IF
    // Limit to avoid value out of array range
    g_iNumBagPerfTear := LIMIT(0,g_iNumBagPerfTear,C_iMaxBagPerfTear) ;

    IF gstCycA[1].CycManTimSet.CmdMov THEN
      g_iArrayBagPerfTear := g_iArrayBagPerfTearNul ;
      gA[1].Cmd_PhaseOffset := 0 ;
      g_iCountPerfShift[1] := 0 ;
      g_iCountPerfShift[2] := 0 ;
    END_IF;

    IF (g_iCountPerfShift[1] > 0)     AND
       EDGENEG(g_bPerfInMatchedSpeed) AND
       g_bMachineRun                  AND
       NOT(gRun_Stop)                 OR
       bTest_[1]                      THEN
       bTest_[1] := 0 ;
      FOR iIndex := g_iNumBagPerfTear-1 TO 1 BY -1 DO
        g_iArrayBagPerfTear[iIndex+1] := g_iArrayBagPerfTear[iIndex] ;
      END_FOR
      g_iArrayBagPerfTear[1] := 0 ;
    END_IF

    IF gA[1].Cmd_PhaseOffset THEN
      g_iCountPerfShift[1] := g_iCountPerfShift[1] + 1 ;
      g_iCountPerfShift[2] := g_iCountPerfShift[1] ;
      IF g_bPerfShiftPos THEN
        g_iArrayBagPerfTear[1] := 1 ;
      ELSE
        g_iArrayBagPerfTear[1] := -1 ;
      END_IF
      g_bPerfShiftPos := 0 ;
    END_IF

    (************************ AXIS PHASE CONTROL (Inches) **********************)
    MC_BR_Phasing_0.Slave:=gA[11].Ident;
    IF gA[1].Ind_SynchronizedMotion AND gA[11].Ind_SynchronizedMotion AND NOT(gstCycA[1].CycManTimSet.bSCyc) AND st_TON_0.Q THEN
      MC_BR_Phasing_0.Enable:=1;
    ELSE;
      MC_BR_Phasing_0.Enable:=0;
    END_IF;
    IF gA[1].Cmd_PhaseOffset  AND NOT(gstCycA[1].CycManTimSet.bSCyc) THEN
      MC_BR_Phasing_0.InitData:=1;
      gA[1].Cmd_PhaseOffset:=0;
      // Calculation new phase Drum/Master
      rTemp_[4] := gA[1].SP_PhaseOffset/gA[11].InchPerDeg ;
      rTemp_[5] := gRecipeActive.rPerf_PhasMasterDeg + rTemp_[4] ;
      gRecipeActive.rPerf_PhasMasterDeg := H_FC_Modulus (IN_rMod := 360, IN_rVar := rTemp_[5]) ;
      rTest_[0] := rTest_[0] + 1 ;
    ELSE
      MC_BR_Phasing_0.InitData:=0;
    END_IF
    MC_BR_Phasing_0.ApplicationMode     := mcMASTER_DISTANCE_BASED;
    MC_BR_Phasing_0.Shift               := gA[1].SP_PhaseOffset*gA[9].UnitsPerInch;
    MC_BR_Phasing_0.Velocity            := 6*gA[11].AxisPeriod/60;
    MC_BR_Phasing_0.Acceleration        := gA[11].SP_Decel;
    //MC_BR_Phasing_0.ApplicationDistance := 0.8*gA[9].AxisPeriod;
    MC_BR_Phasing_0.ApplicationDistance := 0.5*gA[9].AxisPeriod;
    MC_BR_Phasing_0.ShiftMode           := mcRELATIVE;
    MC_BR_Phasing_0();

    (************************ AXIS PHASE CONTROL (Inches) TIMING SETTING **********************)
    IF gstCycA[1].CycManTimSet.bSCyc THEN
      IF gA[1].Cmd_ManuTimSetPlus THEN
        rAxisTimSet_SP_Vel := gr_rAxisTimSet_SP_Vel*gA[9].AxisPeriod/60 / (gA[11].rRSynNum/gA[11].rRSynDen) ;
      ELSE
        rAxisTimSet_SP_Vel := - gr_rAxisTimSet_SP_Vel*gA[9].AxisPeriod/60 / (gA[11].rRSynNum/gA[11].rRSynDen) ;
      END_IF
        rAxisTimSet_SP_Acc := gr_rAxisTimSet_SP_Acc*gA[9].AxisPeriod/60/60 ;
    END_IF

    MC_BR_Phasing_1.Slave                  := gA[11].Ident;
    MC_BR_Phasing_1.Enable                 := gstCycA[1].CycManTimSet.bCyc ;
    MC_BR_Phasing_1.InitData               := gstCycA[1].CycManTimSet.bSCyc ;
    MC_BR_Phasing_1.PerformVelocityControl := gstCycA[1].CycManTimSet.CmdMov ;
    MC_BR_Phasing_1.Velocity               := rAxisTimSet_SP_Vel ;
    MC_BR_Phasing_1.Acceleration           := rAxisTimSet_SP_Acc ;
    MC_BR_Phasing_1.ApplicationMode        := mcVELOCITY_CONTROL ;
    MC_BR_Phasing_1();
    st_TON_0(IN:=NOT(MC_BR_Phasing_1.Enable),PT:=T#100ms) ;

    IF NOT(gstCycA[1].CycManTimSet.CmdMov) AND
       MC_BR_Phasing_1.ShiftAttained       OR
       NOT(gstCycA[1].CycManTimSet.bCyc)   OR
       MC_BR_Phasing_1.Error               AND
       1                                   THEN
      gstCycA[1].CycManTimSet.CmdStop := 0 ;
    END_IF
  END_IF
END_PROGRAM
```

#### A11_BasicInit.st
```iecst
(********************************************************************
 * COPYRIGHT -- Microsoft
 ********************************************************************
 * Program: A11_Basic
 * File: A11_BasicInit.st
 * Author: pkiel
 * Created: July 22, 2011
 ********************************************************************
 * Implementation of program A11_Basic
 ********************************************************************)

PROGRAM _INIT

	(* Axis Setpoint Variables *)
		gA[11].SP_MotorPPR := 36000;
		gA[11].SP_GearBoxInput:= 1;
		gA[11].SP_GearBoxOutput:= 1;
		gA[11].AxisPeriod := (gA[11].SP_MotorPPR*gA[11].SP_GearBoxInput/gA[11].SP_GearBoxOutput);
		gA[11].UnitsPerDeg := gA[11].AxisPeriod/360;
		gA[11].SP_Accel := 0.2*gA[11].AxisPeriod;
		gA[11].SP_Decel := 0.4*gA[11].AxisPeriod;
		gA[11].SP_EStopDecel := 3.0*gA[11].AxisPeriod;
		gA[11].SP_FStopDecel := 1.5*gA[11].AxisPeriod;
		gA[11].HomeVelocity:=12*gA[11].AxisPeriod/60.0;
    gA[11].rSP_CorPosVel := 0.0 ;
    gA[11].rSP_CorPosVel := 0.0 ;
    gA[11].rSP_OverrideV := 1.0 ;
    gA[11].rSP_OverrideA := 1.0 ;

    FOR iIndex := 0 TO C_iMaxBagPerfTear DO
      g_iArrayBagPerfTearNul[iIndex] := 0 ;
    END_FOR ;

	(* access master axis *)
		AxisErrorNcAccess := ncaccess(ncACP10MAN, ADR('Axis11'), ADR(gA[11].Ident));

	(* Trigger Initialization Of ModPosition *)
		InitModPosition:=1;

END_PROGRAM
```

- Program Logical/BagMachine_Section/Perf/Axis11_VirtualAxis/A11_Control (IEC) - Servo Control (no source held here)

### Program Logical/BagMachine_Section/Perf/Axis11_VirtualAxis/A11_Automat (IEC) - Cam Automat

#### A11_Automat.var - Local variables
```iecst
(********************************************************************
 * COPYRIGHT -- Microsoft
 ********************************************************************
 * Program: A11_Automat
 * File: A11_Automat.var
 * Author: pkiel
 * Created: July 22, 2011
 ********************************************************************
 * Local variables of program A11_Automat
 ********************************************************************)
VAR
  AutData : MC_AUTDATA_TYP;
  AutomatStart : BOOL;
  ErrorID : UINT;
  MasterParID : UINT;
  MC_BR_AutControl_0 : MC_BR_AutControl;
  MC_BR_InitMasterParIDTransfer_0 : MC_BR_InitMasterParIDTransfer;
  ParID_Ready : BOOL;
  PositionMOD : DINT;
  PositionOffset : DINT;
  SlaveStartOffset : REAL;
  Synch_Request : BOOL;
  usiMemoStat : USINT;
  InMatched : BOOL ;
  MatchedSpeed_Inch : REAL ;
  rTempPosA1_Inch   : REAL ;
  MasterOffset : REAL ;
  Value1 : DINT ;
  Value2 : DINT ;

END_VAR
```

### CamProfTest.cam
```
CamProfile (NcSwId=ACP10, MasterAxisVelocity=1, MasterAxisAcceleration=0, DefaultCurveType=Polynomial5, MathematicalNotation=true)
  FixPoint (x=360, IsMathX=true, y=180, IsDefinedDy=true, Dy=0.5, IsMathDy=true, IsDefinedDdy=false, Ddy=0, IsMathDdy=true, IsDefinedDddy=false, Dddy=0, IsMathDddy=true)
  Synchronline:
    LeftBoundary (IsFix=true, x=0, IsMathX=true, y=0)
    RightBoundary (IsFix=true, x=120, IsMathX=true, y=60)
    Gradient (Numerator=1, Denominator=2, IsMath=false, IsFix=false)
  Curve (Type=Polynomial5)
    LeftBoundary (IsDefinedDdy=false, Ddy=0, IsMathDdy=true, IsDefinedDddy=false, Dddy=0, IsMathDddy=true)
    RightBoundary (IsDefinedDdy=false, Ddy=0, IsMathDdy=true, IsDefinedDddy=false, Dddy=0, IsMathDddy=true)
    Spline3 (IsContinuous4Derivative=false, IsDefinedSaddlePoint=false, IsDefinedLineAs2ndSegment=false, IsDefinedSlopeOfLine=false, SlopeOfLine=0, IsMathSlopeOfLine=true)
    Supremum (y=1.7e+308, Dy=1.7e+308, IsMathDy=true, Ddy=1.7e+308, IsMathDdy=true, Dddy=1.7e+308, IsMathDddy=true)
    Infimum (y=-1.7e+308, Dy=-1.7e+308, IsMathDy=true, Ddy=-1.7e+308, IsMathDdy=true, Dddy=-1.7e+308, IsMathDddy=true)
  Cam (LeftBoundaryIndex=0, RightBoundaryIndex=1)
    Supremum (y=1.7e+308, Dy=1.7e+308, IsMathDy=true, Ddy=1.7e+308, IsMathDdy=true, Dddy=1.7e+308, IsMathDddy=true)
    Infimum (y=-1.7e+308, Dy=-1.7e+308, IsMathDy=true, Ddy=-1.7e+308, IsMathDdy=true, Dddy=1.7e+308, IsMathDddy=true)
  ChartExtensions
```

### Perf_Gen.typ
```iecst
(********************************************************************
 * COPYRIGHT -- Microsoft
 ********************************************************************
 * Program: Perf_Gen
 * File: Perf_Gen.typ
 * Author: pkiel
 * Created: July 19, 2011
 ********************************************************************
 * Local data types of program Perf_Gen
 ********************************************************************)

TYPE

  PerfPos : STRUCT

  END_STRUCT;

END_TYPE
```

### Perf_Gen.var
```iecst
(********************************************************************
 * COPYRIGHT -- Microsoft
 ********************************************************************
 * Program: Perf_Gen
 * File: Perf_Gen.var
 * Author: pkiel
 * Created: July 19, 2011
 ********************************************************************
 * Local variables of program Perf_Gen
 ********************************************************************)
VAR RETAIN
	HGW_2StatePB_0 : HGW_2StatePB;
END_VAR
VAR
	InParkPosition : BOOL;
	Perf_PB : BOOL;
	PerfColor_Ind : UINT;
	PerfText_Ind : UINT;
	RepeatMetric : INT;
	SecondKnife_Visibility : UINT;
	TON_0 : TON;
	rTempPosA1_Deg : REAL;
	rMatchSpeedPerf : REAL;
	H_FB_Flash_0 : H_FB_Flash;
  HMI_iEnvBPerfSetUpVisible : INT ;
  HMI_iPerfSetUpVisible : INT ;
END_VAR
```

### Package Logical/BagMachine_Section/FP - Axis

- Program Logical/BagMachine_Section/FP/FP_Gen (IEC) - General Flexo Press control (no source held here)

### Program Logical/BagMachine_Section/FP/FP_Dryer (IEC) - Dryer Control

#### DryerCyclic.st - Cyclic code
```iecst
(********************************************************************
 * COPYRIGHT -- .
 ********************************************************************
 * Program: FP_Dryer
 * File: FP_DryerCyclic.st
 * Author: dominique
 * Created: November 08, 2011
 ********************************************************************
 * Implementation of program FP_Dryer
 ********************************************************************)

PROGRAM _CYCLIC

    // -------------------------------------------------------------------
    // Temperature Sensor Alarme
    g_DRY_bTempSensorAlarm := (g_usiAI_DRY_Pt100_TempStatus = 3) ;

    // -------------------------------------------------------------------
    // Blower On/Off
    IF g_DRY_bBlowerAlarm           OR
       EDGENEG(gI_SS_MainPowerOff ) OR
       NOT(g_bMainPower_OnDelay)    OR
       g_bIndEStop                  THEN
      HMI_Cmd_BlowerOnPB := 0 ;
    END_IF ;

    IF HMI_Cmd_AutoOffDryOnPB THEN
      bQ_CR_DRY_Blower := HMI_Cmd_BlowerOnPB AND
                          g_bMachineRun      AND
                          1                  ;
    ELSE
      bQ_CR_DRY_Blower := HMI_Cmd_BlowerOnPB AND
                          1                  ;
    END_IF ;

    // Output activation
    gQ_CR_DRY_Blower := ( bQ_CR_DRY_Blower OR
                          stTOF_0.Q )      AND
                          NOT(g_bIndEStop) ;

    // HMI Blower PB Texte
    IF HMI_Cmd_BlowerOnPB THEN
      uiBlowerOnPBTxt_Ind := 1 ;
    ELSE
      uiBlowerOnPBTxt_Ind := 0 ;
    END_IF ;
    // HMI Dryer Auto Off PB Texte
    IF HMI_Cmd_AutoOffDryOnPB THEN
      uiAutoOffDryOnPBTxt_Ind := 7 ;
    ELSE
      uiAutoOffDryOnPBTxt_Ind := 6 ;
    END_IF ;

    // -------------------------------------------------------------------
    // Heater On/Off
    bActHeat := NOT(g_DRY_bHeaterAlarm) AND
                g_bMainPower_OnDelay    AND
                HMI_Cmd_BlowerOnPB      AND
                NOT(g_bIndEStop)        AND
                1                       ;

    g_DRY_bActHeat := gRecipeActive.bSelHeaterProd AND
                      bQ_CR_DRY_Blower             AND
                      bActHeat                     ;

    // Heater On delayed
    stTON_0(IN:=gQ_CR_DRY_HeatRegul,PT:=T#7s);
    bInd_NeedCool := stTON_0.Q      OR
                     g_DRY_bActHeat AND
                     stTOF_0.Q      ;

    // Blower Off delayed in oder to cool the Heater when switching Off Dryer
    stTOF_0(IN:=bInd_NeedCool,PT:=T#30s);
    rBlowerTimeRemain := (TIME_TO_REAL(stTOF_0.PT) - TIME_TO_REAL(stTOF_0.ET))/1000.0 ;
    // Blower Time Remaining Visible
    IF stTOF_0.Q             AND
       NOT(g_bMachineRun)    AND
       NOT(bQ_CR_DRY_Blower) THEN
      iTimRemVisible := 0 ;
    ELSE
      iTimRemVisible := 1 ;
    END_IF
    g_DRY_bIndCooling := stTOF_0.Q ;
    IF EDGENEG(gI_SS_MainPowerOff ) AND
       g_DRY_bIndCooling            THEN
      g_DRY_bMemPowerOff := 1 ;
    END_IF
    IF NOT(g_DRY_bIndCooling ) THEN
      g_DRY_bMemPowerOff := 0 ;
      g_DRY_bFlash := 0 ;
    END_IF
    H_FB_Flash_0(IN_bEnable:=g_DRY_bMemPowerOff, IN_rNumFlashPerSec:=2) ;
    g_DRY_bFlash := H_FB_Flash_0.OUT_bFlash ;

    // HMI Heater PB Texte
    IF gRecipeActive.bSelHeaterProd THEN
      uiHeaterOnPBTxt_Ind := 3 ;
    ELSE
      uiHeaterOnPBTxt_Ind := 2 ;
    END_IF ;

    // Dryer activated
    g_bSelDryerProd := gRecipeActive.bSelHeaterProd OR
                       HMI_Cmd_BlowerOnPB           OR
                       bTest                        ;

END_PROGRAM
```

### Program Logical/BagMachine_Section/FP/FP_Heater (IEC) - A new program

#### FP_HeaterCyclic.st - Cyclic code
```iecst
(********************************************************************
 * COPYRIGHT -- .
 ********************************************************************
 * Program: FP_Heater
 * File: FP_HeaterCyclic.st
 * Author: dominique
 * Created: August 22, 2012
 ********************************************************************
 * Implementation of program FP_Heater
 ********************************************************************)

PROGRAM _CYCLIC

//------------------------------------------------------------------
// Lecture sonde de temperature
  rSondeTempRegTDegC[1] := INT_TO_REAL(gAI_DRY_Pt100_Temp) / 10.0 ;
  rSondeTempRegTDegF[1] := rSondeTempRegTDegC[1] * 9/5 + 32 ;

  // -------------------------------------------------------------------
  // Temperature Sensor Alarme
  g_DRY_bTempSensorAlarm := (g_usiAI_DRY_Pt100_TempStatus = 3) ;

  // Limit operator Setpoint
  gRecipeActive.rHeatSPDegF := LIMIT(rBornInfConsTempChauf[1],gRecipeActive.rHeatSPDegF,rBornSupConsTempChauf[1]) ;

  // Parametre mesure de temperature du regulateur
  IF g_DRY_bActHeat AND NOT(g_DRY_bTempSensorAlarm) AND NOT(g_bIndEStop) THEN
    rMesTempRegTChauf[1] := rSondeTempRegTDegF[1] ;
  ELSE
    rMesTempRegTChauf[1] := gRecipeActive.rHeatSPDegF ;
  END_IF;

  // Calcul periode echantillonnage appel PID, en s
  // TSI#cycleTime : Temps de cyle de la tache cyclique d appel du regulateur, en ms ( normalmement = 30ms )
  iiRegTChauf_TC[1] := 20 ;
  // Periode appel boucle PID
  rRegTChauf_T[1] := 2 ;

  // Valeur filtree de l'erreur
  // Y = 1/(1+t/T)E + 1/(1+T/t)Y_1
  IF ( rRegTChauf_T[1] <> 0 ) AND
     ( rPT1_t <> 0 )          THEN
    rRegTChauf_ErrF_1[1] := rRegTChauf_ErrF[1] ;
    rRegTChauf_ErrF[1] := ( 1/(1+rPT1_t/rRegTChauf_T[1]) * rRegTChauf_Err[1] + 1/(1+rRegTChauf_T[1]/rPT1_t) * rRegTChauf_ErrF_1[1] ) ;
  END_IF;

  // Appel du PID tout les n cycles PWM
  IF iCptSeuilAppelRegTChauf[1] >= iSeuilAppelPID_RegTChauf[1] THEN
    // Calcul nouvelle erreur
    rRegTChauf_Err[1] := ( gRecipeActive.rHeatSPDegF - rMesTempRegTChauf[1] ) ;
    // Calcul terme proportionnel
    rRegTChauf_TP[1] := rPIDRegTChaufKP[1] * rRegTChauf_Err[1] ;
    // Calcul terme Integral
    IF rPIDRegTChaufKI[1] <> 0.0 THEN  // Traitement cas division par 0
      rRegTChauf_TI[1] := rRegTChauf_TI_1[1] + rRegTChauf_T[1] * 1/rPIDRegTChaufKI[1] * rRegTChauf_Err[1] ;
    ELSE
      rRegTChauf_TI[1] := 0 ;
    END_IF;
    // Init terme Integral sur desactivation regul
    IF g_bIndEStop OR rRegTChauf_TI[1] < 0 OR rRegTChauf_TI_1[1] < 0 OR g_DRY_bTempSensorAlarm THEN
      rRegTChauf_TI[1]   := 0 ;
      rRegTChauf_TI_1[1] := 0 ;
    END_IF;
    // Limitation val sup terme Integral lorsque sortie saturee
    IF rRegTChauf_YPC[1] >= 100 THEN
      rRegTChauf_TI[1] := rRegTChauf_TI_1[1] ;
    END_IF;
    rRegTChauf_TI_1[1] := rRegTChauf_TI[1] ;
    // Calcul terme Derive
    IF rRegTChauf_T[1] <> 0.0 THEN  // Traitement cas division par 0
      rDiff_ErrF[1] := ( rRegTChauf_ErrF[1] - rRegTChauf_Err_1[1] ) ;
      rRegTChauf_TD[1] := 1/rRegTChauf_T[1] * rPIDRegTChaufKD[1] * rDiff_ErrF[1] ;
      // Memo erreur filtree
      rRegTChauf_Err_1[1] := rRegTChauf_ErrF[1] ;
    ELSE
      rRegTChauf_TD[1] := 0 ;
    END_IF;
    // Calcul sortie
    rRegTChauf_Y[1] := rRegTChauf_TP[1] + rRegTChauf_TI[1] + rRegTChauf_TD[1] ;
    // Conversion sortie en %
    IF rBornSupConsTempChauf[1] <> 0.0 THEN  // Traitement cas division par 0
      rRegTChauf_YPC[1] := rRegTChauf_Y[1] /rBornSupConsTempChauf[1] * 100 ;
    ELSE
      rRegTChauf_YPC[1] := 0 ;
    END_IF;
    IF rRegTChauf_YPC[1] > 100 THEN
      rRegTChauf_YPC[1] := 100 ;
    END_IF;
    IF rRegTChauf_YPC[1] < 0 OR g_DRY_bTempSensorAlarm OR g_bIndEStop OR NOT(g_DRY_bActHeat) THEN
      rRegTChauf_YPC[1] := 0 ;
    END_IF;
  END_IF;

  // Appel bloc PID
  // Incrementation et remise a zero du compteur d'appel du PID
  iSeuilAppelPID_RegTChauf[1] := 100 ; // Pour une tache interruptive de 20ms 100x20 = 2000ms = 2s
  iCptSeuilAppelRegTChauf[1]  := iCptSeuilAppelRegTChauf[1]  + 1  ;
  IF iCptSeuilAppelRegTChauf[1] > iSeuilAppelPID_RegTChauf[1] THEN
    iCptSeuilAppelRegTChauf[1] := 0 ;
  END_IF;

  // Parametres du PWM
  LCRPWM_0[1].enable      := 1 ;
  LCRPWM_0[1].x           := rRegTChauf_YPC[1] ;
  LCRPWM_0[1].max_value   := 100.0 ;
  LCRPWM_0[1].min_value   := 0.0 ;
  LCRPWM_0[1].t_min_pulse := iiRegTChauf_TC[1] / 1000 ;
  LCRPWM_0[1].t_period    := rRegTChauf_T[1] ;
  LCRPWM_0[1]() ;

  // Activation de la sortie regulee
  IF g_DRY_bActHeat AND NOT(g_DRY_bTempSensorAlarm) AND NOT(g_bIndEStop) THEN
    bImdoRT_ActChauf[1] := LCRPWM_0[1].pulse AND NOT(bTest) ;
  ELSE
    bImdoRT_ActChauf[1] := 0 ;
  END_IF;
  gQ_CR_DRY_HeatRegul := bImdoRT_ActChauf[1] ;

  // Calcul pic de chauffe a l'activation du chauffage
  IF EDGEPOS(g_DRY_bActHeat) THEN
    bImpulsDemarSech := 1 ;
  END_IF ;
  IF rSondeTempRegTDegF[1] >= gRecipeActive.rHeatSPDegF - rDeltaTStopPicChauf THEN
    bImpulsDemarSech := 0 ;
  END_IF ;

  // Batterie de chauffe TOR
  IF gRecipeActive.rHeatSPDegF > rSeuilConsTempActBattTOR OR
    bImpulsDemarSech                                      THEN
    gQ_CR_DRY_HeatContinu := g_DRY_bActHeat AND NOT(bTest);
  ELSE
    gQ_CR_DRY_HeatContinu := 0 ;
  END_IF ;

  // Conversion for trending
  IF ( gInchMetric_Ind = 2 ) THEN
    rTrendActTempRegT[1]   := rSondeTempRegTDegC[1] ;
    rTrendSetPTempRegT[1]  := (gRecipeActive.rHeatSPDegF-32) * 5/9 ;
    rTrendRegTChauf_Err[1] := (rRegTChauf_Err[1]-32) * 5/9 ;
  ELSE
    rTrendActTempRegT[1]   := rSondeTempRegTDegF[1] ;
    rTrendSetPTempRegT[1]  := gRecipeActive.rHeatSPDegF ;
    rTrendRegTChauf_Err[1] := rRegTChauf_Err[1] ;
  END_IF;

END_PROGRAM
```

- Data object Logical/BagMachine_Section/FP/Axis2/A2_Init (Ax) - Servo Axis Initialization File (no source held here)

### Data object Logical/BagMachine_Section/FP/Axis2/A2_Par (Apt) - Servo Axis Parameter File

#### A2_Par.apt
```
AcoposParameterTable:
  Root Parameters:
    110 = ncSW_OFF (Name=CMD_SIMULATION)  // Simulation mode: Command
    128 = 1 (Name=SGEN_SW_END_IGNORE)  // SGEN_SW_END_IGNORE
    Axis Parameter Identification Induction Motor:
      General Parameters:
        30 = 1 (Name=MOTOR_TYPE)  // Motor: Type
        31 = 515 (Name=MOTOR_COMPATIBILITY)  // Motor: Software compatibility
        46 = 1 (Name=MOTOR_WIND_CONNECT)  // Motor: Winding connection
        62 = 0.109 (Name=MOTOR_INERTIA, Unit=kgm²)  // Motor: Moment of inertia
        849 = 0 (Name=MOTOR_TAU_THERM, Unit=s)  // Motor: Thermal time constant
      Brake Parameters:
        42 = 0 (Name=MOTOR_BRAKE_CURR_RATED, Unit=A)  // Motor holding brake: Rated current
        43 = 0 (Name=MOTOR_BRAKE_TORQ_RATED, Unit=Nm)  // Motor holding brake: Rated torque
        44 = 0 (Name=MOTOR_BRAKE_ON_TIME, Unit=s)  // Motor holding brake: Engaging delay
        45 = 0 (Name=MOTOR_BRAKE_OFF_TIME, Unit=s)  // Motor holding brake: Release delay
      Thermo Sensor Parameters:
        64 = 391 (Name=MOTOR_TEMPSENS_PAR1)  // Temperature sensor: Parameter 1
        65 = 1492 (Name=MOTOR_TEMPSENS_PAR2)  // Temperature sensor: Parameter 2
        66 = -30 (Name=MOTOR_TEMPSENS_PAR3)  // Temperature sensor: Parameter 3
        67 = 12.01 (Name=MOTOR_TEMPSENS_PAR4)  // Temperature sensor: Parameter 4
        68 = 45.98 (Name=MOTOR_TEMPSENS_PAR5)  // Temperature sensor: Parameter 5
        69 = 75.71 (Name=MOTOR_TEMPSENS_PAR6)  // Temperature sensor: Parameter 6
        70 = 102.2 (Name=MOTOR_TEMPSENS_PAR7)  // Temperature sensor: Parameter 7
        71 = 126.41 (Name=MOTOR_TEMPSENS_PAR8)  // Temperature sensor: Parameter 8
        72 = 148.88 (Name=MOTOR_TEMPSENS_PAR9)  // Temperature sensor: Parameter 9
        73 = 170 (Name=MOTOR_TEMPSENS_PAR10)  // Temperature sensor: Parameter 10
        74 = 100 (Name=MOTOR_WIND_TEMP_MAX, Unit=°C)  // Temperature sensor: Limit temperature
      Result Parameters of Parameter Identification:
        47 = 2 (Name=MOTOR_POLEPAIRS)  // Motor: Number of pole-pairs
        48 = 322 (Name=MOTOR_VOLTAGE_RATED, Unit=V)  // Motor: Rated voltage
        49 = 0 (Name=MOTOR_VOLTAGE_CONST, Unit=mV*min)  // Motor: Voltage constant
        50 = 1000 (Name=MOTOR_SPEED_RATED, Unit=1/min)  // Motor: Rated speed
        51 = 8000 (Name=MOTOR_SPEED_MAX, Unit=1/min)  // Motor: Maximum speed
        52 = 162.34 (Name=MOTOR_TORQ_STALL, Unit=Nm)  // Motor: Stall torque
        53 = 162.34 (Name=MOTOR_TORQ_RATED, Unit=Nm)  // Motor: Rated torque
        54 = 577.34 (Name=MOTOR_TORQ_MAX, Unit=Nm)  // Motor: Peak torque
        55 = 0 (Name=MOTOR_TORQ_CONST, Unit=Nm/A)  // Motor: Torque constant
        56 = 40.69 (Name=MOTOR_CURR_STALL, Unit=A)  // Motor: Stall current
        57 = 40.69 (Name=MOTOR_CURR_RATED, Unit=A)  // Motor: Rated current
        58 = 238.47 (Name=MOTOR_CURR_MAX, Unit=A)  // Motor: Peak current
        59 = 0 (Name=MOTOR_WIND_CROSS_SECT, Unit=mm²)  // Motor: Line cross section
        60 = 0.1542 (Name=MOTOR_STATOR_RESISTANCE, Unit=Ohm)  // Motor: Stator resistance
        61 = 0.00180 (Name=MOTOR_STATOR_INDUCTANCE, Unit=Henry)  // Motor: Stator inductance
        63 = 0 (Name=MOTOR_COMMUT_OFFSET, Unit=rad)  // Motor: Commutation offset
        76 = 0.10915 (Name=MOTOR_ROTOR_RESISTANCE, Unit=Ohm)  // Motor: Rotor resistance
        77 = 0.00180 (Name=MOTOR_ROTOR_INDUCTANCE, Unit=Henry)  // Motor: Rotor inductance
        78 = 0.0527 (Name=MOTOR_MUTUAL_INDUCTANCE, Unit=Henry)  // Motor: Mutual inductance
        79 = 18.5 (Name=MOTOR_MAGNETIZING_CURR, Unit=A)  // Motor: Magnetizing current
```

### Program Logical/BagMachine_Section/FP/Axis2/A2_Control (IEC) - Servo Control

#### A2_Control.var
```iecst
(********************************************************************
 * COPYRIGHT -- Microsoft
 ********************************************************************
 * Program: A2_Control
 * File: A2_Control.var
 * Author: Dominique
 * Created: October 15, 2011
 ********************************************************************
 * Local variables of program A2_Control
 ********************************************************************)
VAR
	HGW_ChangeReal_0 : HGW_ChangeReal;
	HGW_RelativeChangeReal_0 : H_FB_RelativeChangeLimitReal1;
	HGW_Toggle_0 : HGW_Toggle;
	Synch_Permissive : BOOL;
	TOF_0 : TOF;
	TON_0 : TON;
  rIncrOffsetAxeRun_Inch : REAL ;
  rPoub : ARRAY[0..5] OF REAL ;
  bCmd_ManuTimSet : BOOL ;

  HMI_Cmd_ManuTimSetPlus : BOOL ;
  bLockSP_OffsetPrintRol : BOOL ;
END_VAR
```

#### A2_ControlCyclic.ld
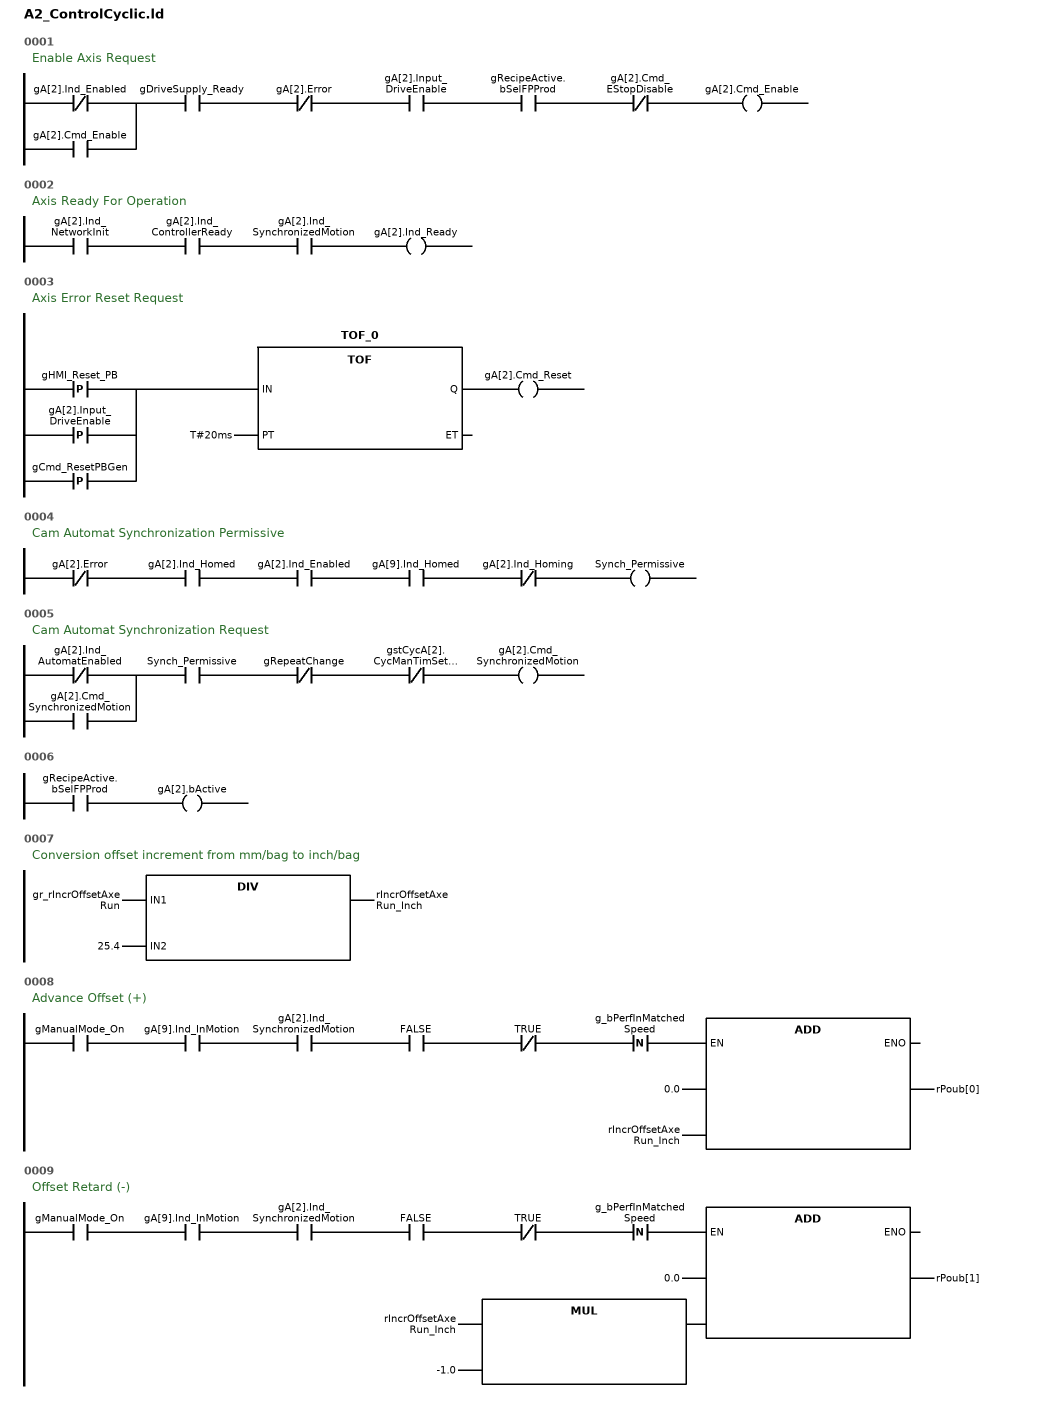
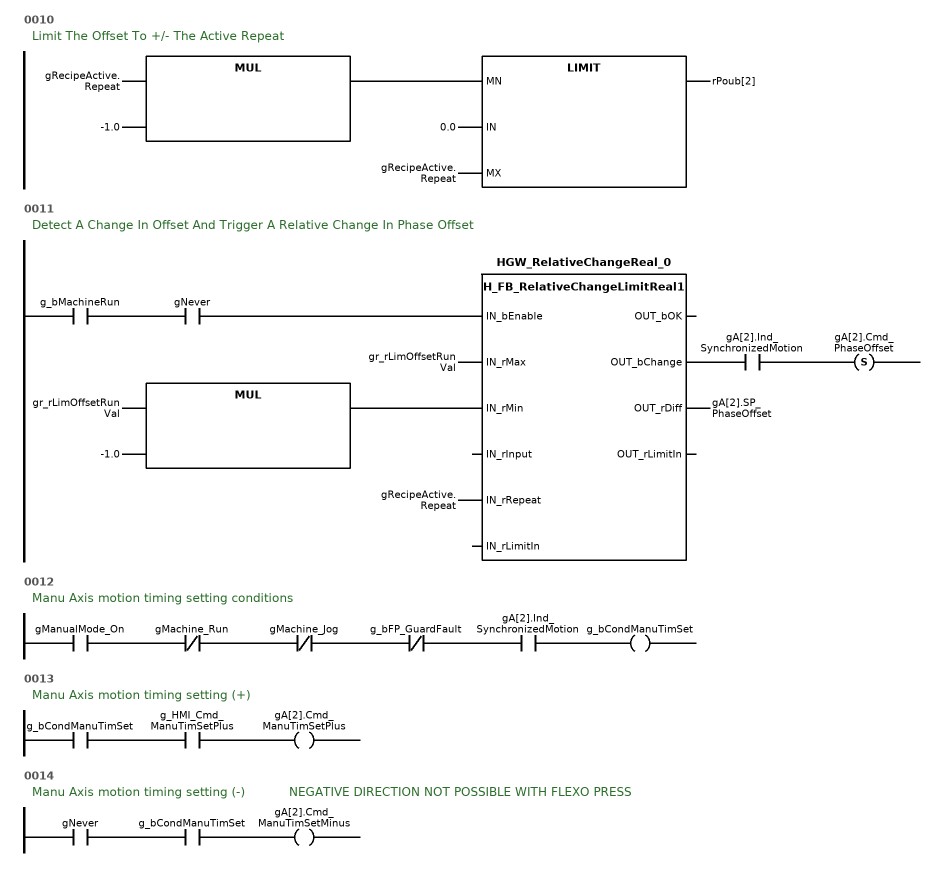
Ladder, written as Structured Text:
```iecst
(********************************************************************
 * COPYRIGHT -- Microsoft
 ********************************************************************
 * Program: A7_Control
 * File: A7_ControlCyclic.ld
 * Author: pkiel
 * Created: July 13, 2011
 ********************************************************************
 * Implementation of program A7_Control
 ********************************************************************)

PROGRAM _CYCLIC
VAR
    _e1 : R_TRIG;
    _e2 : R_TRIG;
    _e3 : R_TRIG;
    _e4 : F_TRIG;
    _e5 : F_TRIG;
END_VAR
(* Network 1: Enable Axis Request *)
gA[2].Cmd_Enable := (NOT gA[2].Ind_Enabled OR gA[2].Cmd_Enable) AND gDriveSupply_Ready AND NOT gA[2].Error AND gA[2].Input_DriveEnable AND gRecipeActive.bSelFPProd AND NOT gA[2].Cmd_EStopDisable;

(* Network 2: Axis Ready For Operation *)
gA[2].Ind_Ready := gA[2].Ind_NetworkInit AND gA[2].Ind_ControllerReady AND gA[2].Ind_SynchronizedMotion;

(* Network 3: Axis Error Reset Request *)
_e1(CLK := gHMI_Reset_PB);
_e2(CLK := gA[2].Input_DriveEnable);
_e3(CLK := gCmd_ResetPBGen);
TOF_0(IN := _e1.Q OR _e2.Q OR _e3.Q, PT := T#20ms);
gA[2].Cmd_Reset := TOF_0.Q;

(* Network 4: Cam Automat Synchronization Permissive *)
Synch_Permissive := NOT gA[2].Error AND gA[2].Ind_Homed AND gA[2].Ind_Enabled AND gA[9].Ind_Homed AND NOT gA[2].Ind_Homing;

(* Network 5: Cam Automat Synchronization Request *)
gA[2].Cmd_SynchronizedMotion := (NOT gA[2].Ind_AutomatEnabled OR gA[2].Cmd_SynchronizedMotion) AND Synch_Permissive AND NOT gRepeatChange AND NOT gstCycA[2].CycManTimSet.CmdExeStop;

(* Network 6 *)
gA[2].bActive := gRecipeActive.bSelFPProd;

(* Network 7: Conversion offset increment from mm/bag to inch/bag *)
rIncrOffsetAxeRun_Inch := gr_rIncrOffsetAxeRun / 25.4;

(* Network 8: Advance Offset (+) *)
_e4(CLK := g_bPerfInMatchedSpeed);
(* never executed: rPoub[0] := 0.0 + rIncrOffsetAxeRun_Inch; *)

(* Network 9: Offset Retard (-) *)
_e5(CLK := g_bPerfInMatchedSpeed);
(* never executed: rPoub[1] := 0.0 + (rIncrOffsetAxeRun_Inch * -1.0); *)

(* Network 10: Limit The Offset To +/- The Active Repeat *)
rPoub[2] := LIMIT(MN := gRecipeActive.Repeat * -1.0, IN := 0.0, MX := gRecipeActive.Repeat);

(* Network 11: Detect A Change In Offset And Trigger A Relative Change In Phase Offset *)
HGW_RelativeChangeReal_0(IN_bEnable := g_bMachineRun AND gNever, IN_rMax := gr_rLimOffsetRunVal, IN_rMin := gr_rLimOffsetRunVal * -1.0, IN_rRepeat := gRecipeActive.Repeat);
IF HGW_RelativeChangeReal_0.OUT_bChange AND gA[2].Ind_SynchronizedMotion THEN
    gA[2].Cmd_PhaseOffset := TRUE;
END_IF;
gA[2].SP_PhaseOffset := HGW_RelativeChangeReal_0.OUT_rDiff;

(* Network 12: Manu Axis motion timing setting conditions *)
g_bCondManuTimSet := gManualMode_On AND NOT gMachine_Run AND NOT gMachine_Jog AND NOT g_bFP_GuardFault AND gA[2].Ind_SynchronizedMotion;

(* Network 13: Manu Axis motion timing setting (+) *)
gA[2].Cmd_ManuTimSetPlus := g_bCondManuTimSet AND g_HMI_Cmd_ManuTimSetPlus;

(* Network 14: Manu Axis motion timing setting (-)           NEGATIVE DIRECTION NOT POSSIBLE WITH FLEXO PRESS *)
gA[2].Cmd_ManuTimSetMinus := gNever AND g_bCondManuTimSet;
END_PROGRAM
```

### Program Logical/BagMachine_Section/FP/Axis2/A2_Automat (IEC) - Cam Automat

#### A2_AutomatCyclic.st - Cyclic code
```iecst
(********************************************************************
 * COPYRIGHT -- Microsoft
 ********************************************************************
 * Program: A2_Automat
 * File: A2_AutomatCyclic.st
 * Author: Dominique
 * Created: October 15, 2011
 ********************************************************************
 * Implementation of program A2_Automat
 ********************************************************************)

PROGRAM _CYCLIC

  IF (gRecipeActive.iPrintUp <= 0.0)         OR
     (gRecipeActive.iNumToothGearPrint <= 0) OR
     (g_rZGearRepFP <= 0.0)                  THEN
    RETURN ;
  END_IF

  // Synchro ratio Master/Slave
  rPrintUp := INT_TO_REAL(gRecipeActive.iPrintUp) ; // Number of pictures per round of printing cylinder
     // Master = Virtuel or Tearing
     gA[2].rRSynNum := gRecipeActive.iNumToothGearPrint ;
     gA[2].rRSynDen := g_rZGearRepFP * rPrintUp ;

  // Signal synchro Holding axis
  MC_BR_AutControl_0.Signal1 := gA[3].Ind_bSynchroOK               AND
                                NOT(gstCycA[2].CycManTimSet.bSCyc) ;

  // FP timing setting
  IF EDGEPOS(gstCycA[2].CycManTimSet.CmdSynchroOn) THEN
    MC_BR_AutControl_0.Signal2 := 1 ;
    MC_BR_AutControl_0.Signal3 := 0 ;
    MC_BR_AutControl_0.Signal4 := 0 ;
  END_IF
  IF EDGENEG(gstCycA[2].CycManTimSet.CmdSynchroOn) THEN
    MC_BR_AutControl_0.Signal2 := 0 ;
    IF gA[3].Ind_bSynchroOK THEN
      MC_BR_AutControl_0.Signal3 := 1 ;
      MC_BR_AutControl_0.Signal4 := 0 ;
    ELSE
      MC_BR_AutControl_0.Signal4 := 1 ;
      MC_BR_AutControl_0.Signal3 := 0 ;
    END_IF
  END_IF

  // A2 Synchro OK indicator
  gstCycA[2].CycManTimSet.bSynchroOkSlavA[2] := ( MC_BR_AutControl_0.ActualStateIndex = 4 )  AND
                                                gA[2].Ind_SynchronizedMotion AND ParID_Ready ;

(**** STRAIGHT GEARED CAM AUTOMAT WITH ABSOLUTE PHASE SYNCHRONIZATION FOR DRUM ***)
  Synch_Request := gA[2].Cmd_SynchronizedMotion;
  IF (Synch_Request AND NOT ParID_Ready) THEN
    MC_BR_InitMasterParIDTransfer_0.Master:= gA[9].Ident ;
    MC_BR_InitMasterParIDTransfer_0.Slave:= gA[2].Ident ;
    MC_BR_InitMasterParIDTransfer_0.MasterParID:= 412 ; // ParID 412 = 412: VAX: Position (in case virtual axis)
    MC_BR_InitMasterParIDTransfer_0.SlaveChannel:=0;
    MC_BR_InitMasterParIDTransfer_0.Execute:=TRUE;
    IF (MC_BR_InitMasterParIDTransfer_0.Done) THEN
      MasterParID:=MC_BR_InitMasterParIDTransfer_0.ReceiveParID;
      MC_BR_InitMasterParIDTransfer_0.Execute:=FALSE;
      ParID_Ready:=1;
    ELSIF (MC_BR_InitMasterParIDTransfer_0.Error) THEN
    (*Store ErrorID in a variable,
      ErrorID is reset on falling edge of 'Execute'*)
      ErrorID:=MC_BR_InitMasterParIDTransfer_0.ErrorID;
      ParID_Ready:=0;
      MC_BR_InitMasterParIDTransfer_0.Execute:=FALSE;
    END_IF
  END_IF
  MC_BR_InitMasterParIDTransfer_0();

(**** Initialize Automat Parameters Upon Automat Start Request ****)
  IF (EDGEPOS(ParID_Ready))THEN

    (**** Calculate Slave Start Offset ****)
      MasterOffset := gRecipeActive.Drum_Offset + gRecipeActive.Holding_Offset + gRecipeActive.Tearing_Offset;
      PositionOffset:= REAL_TO_DINT((gA[9].PositionInch-(gA[2].PositionInch-MasterOffset))*1000);
      PositionMOD:= REAL_TO_DINT(gRecipeActive.Repeat*1000);
      SlaveStartOffset:= (DINT_TO_REAL(PositionOffset MOD PositionMOD))/1000;
      IF (SlaveStartOffset >= (0.5*gRecipeActive.Repeat)) THEN
        SlaveStartOffset := SlaveStartOffset - gRecipeActive.Repeat;
      END_IF
      IF (SlaveStartOffset < (-0.5*gRecipeActive.Repeat)) THEN
        SlaveStartOffset := SlaveStartOffset + gRecipeActive.Repeat;
      END_IF

    (*general automat parameter*)
      (*AutData.Master          := gA1.Ident;*)
      AutData.MasterParID        := MasterParID;
      AutData.StartPosition      := 0;
      AutData.StartInterval      := gA[9].AxisPeriod;
      AutData.MaxMasterVelocity  := gr_rMachMaxSpeed_BPM ;

    (*Automat STATE 0 Basis State*)
      AutData.State[0].Event[0].Type      := ncSIGNAL1;
      AutData.State[0].Event[0].Attribute  := ncAT_ONCE;
      AutData.State[0].Event[0].NextState := 3 ;

      AutData.State[0].Event[1].Type      := ncSIGNAL2;
      AutData.State[0].Event[1].Attribute  := ncAT_ONCE;
      AutData.State[0].Event[1].NextState := 4 ;

    (*//Automat STATE 1 Master/Slave Absolute Phase Correction
      AutData.State[1].MasterParID     := MasterParID ;
      AutData.State[1].CamProfileIndex := 16#FFFF;
      AutData.State[1].MasterFactor     := REAL_TO_UDINT(gA[9].AxisPeriod*2);
      AutData.State[1].SlaveFactor     := REAL_TO_UDINT((gA[2].AxisPeriod*2)+(rSlCompDist*gA[2].UnitsPerDeg));
      AutData.State[1].CompMode         := ncOFF;

      AutData.State[1].Event[0].Type      := ncST_END;
      AutData.State[1].Event[0].Attribute := ncST_END;
      AutData.State[1].Event[0].NextState := 3;

    //Automat STATE 2 Master/Slave Transition
      AutData.State[2].MasterParID        := MasterParID ;
      AutData.State[2].CamProfileIndex    := 16#FFFF;
      AutData.State[2].MasterFactor        := REAL_TO_UDINT(gA[9].AxisPeriod/2);
      AutData.State[2].SlaveFactor        := REAL_TO_UDINT(gA[2].AxisPeriod/2);
      AutData.State[2].CompMode            := ncONLYCOMP;
      AutData.State[2].MasterCompDistance := gA[9].AxisPeriod-AutData.State[2].MasterFactor;
      AutData.State[2].SlaveCompDistance  := gA[3].AxisPeriod-AutData.State[2].SlaveFactor;
      AutData.State[2].ExtendedCompLimits := ncOFF;

      AutData.State[2].Event[0].Type      := ncST_END;
      AutData.State[2].Event[0].Attribute  := ncST_END;
      AutData.State[2].Event[0].NextState  := 3;*)

    //Automat STATE 3 Master/Slave Run
      AutData.State[3].MasterParID     := MasterParID ;
      AutData.State[3].CamProfileIndex := 16#FFFF;
      AutData.State[3].MasterFactor     := REAL_TO_UDINT(gA[2].rRSynDen*gA[9].AxisPeriod);
      AutData.State[3].SlaveFactor     := REAL_TO_UDINT(gA[2].rRSynNum*gA[2].AxisPeriod);
      AutData.State[3].CompMode         := ncOFF;

      AutData.State[3].Event[0].Type      := ncST_END;
      AutData.State[3].Event[0].Attribute := ncST_END;
      AutData.State[3].Event[0].NextState := 3;

      AutData.State[3].Event[1].Type      := ncSIGNAL2 ;
      AutData.State[3].Event[1].Attribute := ncAT_ONCE ;
      AutData.State[3].Event[1].NextState := 4 ;

    //Automat STATE 4 Master/Slave Timing setting
      AutData.State[4].CamProfileIndex := 16#FFFF;
      AutData.State[4].MasterFactor    := REAL_TO_UDINT(gA[9].AxisPeriod) ;
      AutData.State[4].SlaveFactor     := REAL_TO_UDINT(gA[2].AxisPeriod) ;
      AutData.State[4].CompMode        := ncOFF;

      AutData.State[4].Event[0].Type      := ncST_END ;
      AutData.State[4].Event[0].Attribute := ncST_END ;
      AutData.State[4].Event[0].NextState := 4 ;

      AutData.State[4].Event[1].Type      := ncST_END+ncNEGATIVE ;
      AutData.State[4].Event[1].Attribute := ncST_END ;
      AutData.State[4].Event[1].NextState := 4 ;

      AutData.State[4].Event[2].Type      := ncSIGNAL3 ;
      AutData.State[4].Event[2].Attribute := ncAT_ONCE ;
      AutData.State[4].Event[2].NextState := 3 ;

      AutData.State[4].Event[3].Type      := ncSIGNAL4 ;
      AutData.State[4].Event[3].Attribute := ncAT_ONCE ;
      AutData.State[4].Event[3].NextState := 0 ;

      MC_BR_AutControl_0.Enable      := 1;
      MC_BR_AutControl_0.AdrAutData  := ADR(AutData);
      MC_BR_AutControl_0.InitAutData := 1;
  END_IF
      (* wait for initialization done or restart *)
      IF ((MC_BR_AutControl_0.AutDataInitialized=1) AND (Synch_Request)) THEN
        MC_BR_AutControl_0.InitAutData := 0;
        MC_BR_AutControl_0.Enable :=1;
        AutomatStart := 1;;
      END_IF
      (* check if error occured *)
      IF (MC_BR_AutControl_0.ErrorID <> 0) THEN
        MC_BR_AutControl_0.Enable := 0;
      END_IF

  (******************** ENABLE CAM-AUTOMAT **********************)

  IF (AutomatStart) THEN
      MC_BR_AutControl_0.Start := 1;
      AutomatStart := 0;
  END_IF

  IF (NOT Synch_Request) THEN
      MC_BR_AutControl_0.Stop := 1;
      MC_BR_AutControl_0.Start := 0;
      ParID_Ready := 0;
      IF (MC_BR_AutControl_0.Running=0) THEN
        MC_BR_AutControl_0.Enable := 0;
        MC_BR_AutControl_0.Stop := 0;
      END_IF
  END_IF

  gA[2].Ind_AutomatEnabled:=MC_BR_AutControl_0.Enable;
  gA[2].Ind_CurrentAutomatState:=MC_BR_AutControl_0.ActualStateIndex;
  gA[2].Ind_bSynchroOK := (MC_BR_AutControl_0.ActualStateIndex >= 3) AND gA[2].Ind_SynchronizedMotion ; ;

  (********************** MC_AUTCONTROL *************************)
  MC_BR_AutControl_0.Slave:= gA[2].Ident;
  MC_BR_AutControl_0();

END_PROGRAM
```

#### A2_Automat.var - Local variables
```iecst
(********************************************************************
 * COPYRIGHT -- Microsoft
 ********************************************************************
 * Program: A2Automat
 * File: A2Automat.var
 * Author: Dominique
 * Created: October 15, 2011
 ********************************************************************
 * Local variables of program A2Automat
 ********************************************************************)
VAR
	AutData : MC_AUTDATA_TYP;
	AutomatStart : BOOL;
	ErrorID : UINT;
	MasterOffset : REAL;
  MasterParID : UINT;
  uiMasterParID1 : UINT;
	MC_BR_AutControl_0 : MC_BR_AutControl;
  MC_BR_InitMasterParIDTransfer_0 : MC_BR_InitMasterParIDTransfer;
  MC_BR_InitMasterParIDTransfer_1 : MC_BR_InitMasterParIDTransfer;
  ParID_Ready : BOOL;
  ParID_Ready1 : BOOL;
	PositionMOD : DINT;
	PositionOffset : DINT;
	SlaveStartOffset : REAL;
	Synch_Request : BOOL;
  uiSP_MasterParID : UINT;
  uiiSP_Master : UDINT;
  uiiSlaveFactor : UDINT;
  uiiMasterFactor : UDINT;
  usiMemoStat : USINT ;
  iiMasterFactor5 : DINT;
  iiSlaveFactor5  : DINT;
  bCmdSynchroOn : BOOL ;
  bCmdSynchroOff : BOOL ;
  rMaCompDist : REAL ;
  rSPMaPos    : REAL ;
  rOffsetDeg  : REAL ;
  rSlCompDist : REAL ;
  rTemp_      : ARRAY[0..9] OF REAL ;
  rPrintUp    : REAL ;
END_VAR
```

### Program Logical/BagMachine_Section/FP/Axis2/A2_Ref (IEC) - Reference Routine

#### A2_RefCyclic.ld
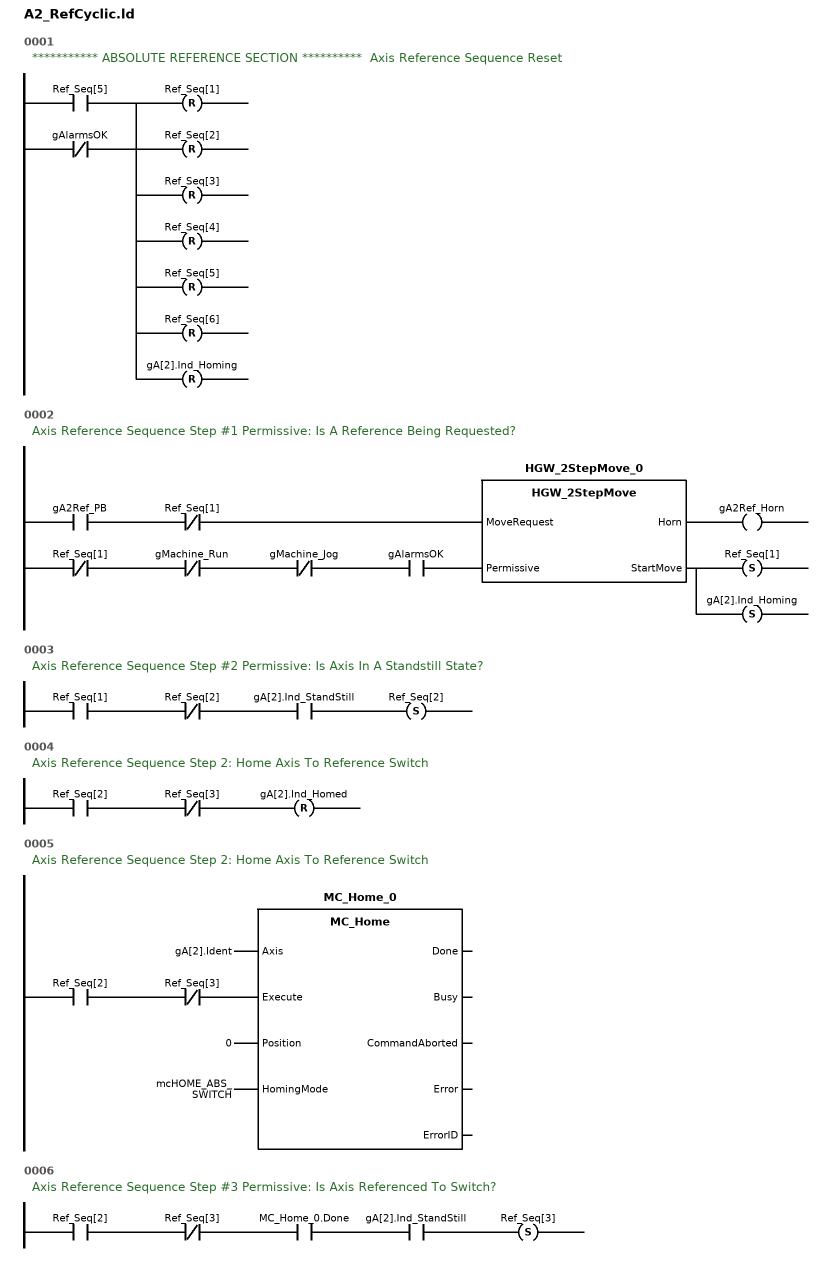
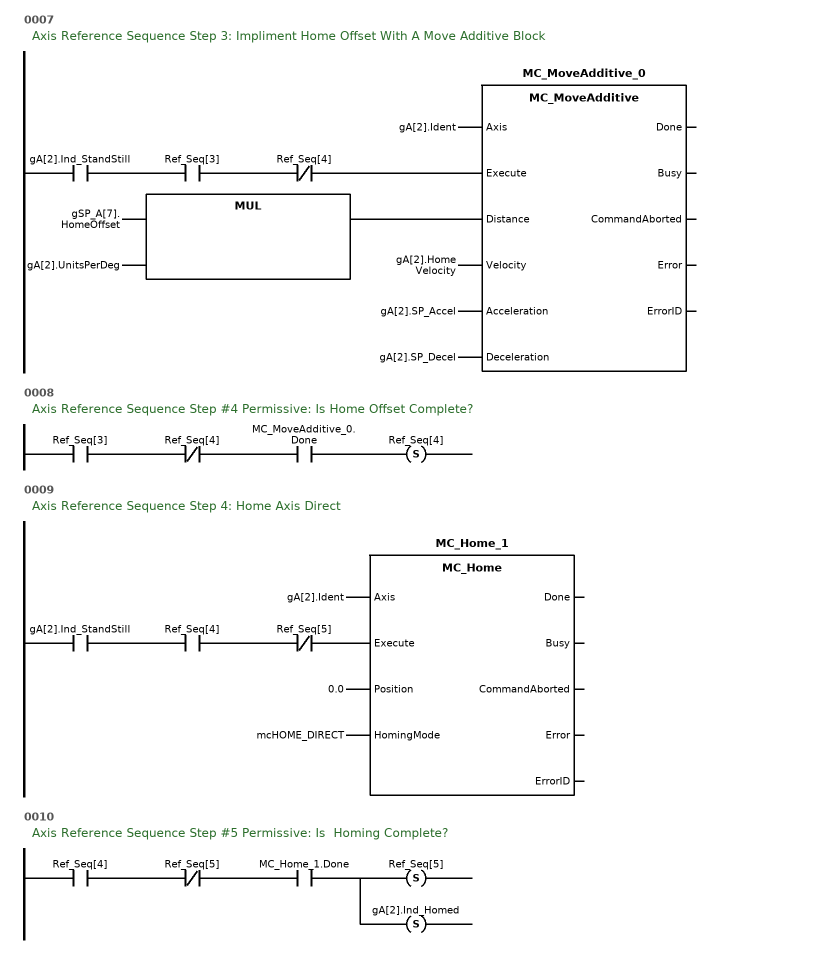
Ladder, written as Structured Text:
```iecst
(********************************************************************
 * COPYRIGHT -- Microsoft
 ********************************************************************
 * Program: A7_Ref
 * File: A7_RefCyclic.ld
 * Author: pkiel
 * Created: July 19, 2011
 ********************************************************************
 * Implementation of program A7_Ref
 ********************************************************************)

PROGRAM _CYCLIC
VAR
    _p1 : BOOL;
    _p2 : BOOL;
END_VAR
(* Network 1: *********** ABSOLUTE REFERENCE SECTION **********  Axis Reference Sequence Reset *)
_p1 := Ref_Seq[5];
IF Ref_Seq[5] OR NOT gAlarmsOK THEN Ref_Seq[1] := FALSE; END_IF;
IF _p1 OR NOT gAlarmsOK THEN
    Ref_Seq[2] := FALSE;
    Ref_Seq[3] := FALSE;
    Ref_Seq[4] := FALSE;
    Ref_Seq[5] := FALSE;
    Ref_Seq[6] := FALSE;
    gA[2].Ind_Homing := FALSE;
END_IF;

(* Network 2: Axis Reference Sequence Step #1 Permissive: Is A Reference Being Requested? *)
HGW_2StepMove_0(MoveRequest := gA2Ref_PB AND NOT Ref_Seq[1], Permissive := NOT Ref_Seq[1] AND NOT gMachine_Run AND NOT gMachine_Jog AND gAlarmsOK);
gA2Ref_Horn := HGW_2StepMove_0.Horn;
IF HGW_2StepMove_0.StartMove THEN
    Ref_Seq[1] := TRUE;
    gA[2].Ind_Homing := TRUE;
END_IF;

(* Network 3: Axis Reference Sequence Step #2 Permissive: Is Axis In A Standstill State? *)
IF Ref_Seq[1] AND NOT Ref_Seq[2] AND gA[2].Ind_StandStill THEN Ref_Seq[2] := TRUE; END_IF;

(* Network 4: Axis Reference Sequence Step 2: Home Axis To Reference Switch *)
IF Ref_Seq[2] AND NOT Ref_Seq[3] THEN gA[2].Ind_Homed := FALSE; END_IF;

(* Network 5: Axis Reference Sequence Step 2: Home Axis To Reference Switch *)
MC_Home_0(Axis := gA[2].Ident, Execute := Ref_Seq[2] AND NOT Ref_Seq[3], Position := 0, HomingMode := mcHOME_ABS_SWITCH);

(* Network 6: Axis Reference Sequence Step #3 Permissive: Is Axis Referenced To Switch? *)
IF Ref_Seq[2] AND NOT Ref_Seq[3] AND MC_Home_0.Done AND gA[2].Ind_StandStill THEN
    Ref_Seq[3] := TRUE;
END_IF;

(* Network 7: Axis Reference Sequence Step 3: Impliment Home Offset With A Move Additive Block *)
MC_MoveAdditive_0(Axis := gA[2].Ident, Execute := gA[2].Ind_StandStill AND Ref_Seq[3] AND NOT Ref_Seq[4], Distance := gSP_A[7].HomeOffset * gA[2].UnitsPerDeg, Velocity := gA[2].HomeVelocity, Acceleration := gA[2].SP_Accel, Deceleration := gA[2].SP_Decel);

(* Network 8: Axis Reference Sequence Step #4 Permissive: Is Home Offset Complete? *)
IF Ref_Seq[3] AND NOT Ref_Seq[4] AND MC_MoveAdditive_0.Done THEN Ref_Seq[4] := TRUE; END_IF;

(* Network 9: Axis Reference Sequence Step 4: Home Axis Direct *)
MC_Home_1(Axis := gA[2].Ident, Execute := gA[2].Ind_StandStill AND Ref_Seq[4] AND NOT Ref_Seq[5], Position := 0.0, HomingMode := mcHOME_DIRECT);

(* Network 10: Axis Reference Sequence Step #5 Permissive: Is  Homing Complete? *)
_p2 := Ref_Seq[4] AND NOT Ref_Seq[5] AND MC_Home_1.Done;
IF Ref_Seq[4] AND NOT Ref_Seq[5] AND MC_Home_1.Done THEN Ref_Seq[5] := TRUE; END_IF;
IF _p2 THEN gA[2].Ind_Homed := TRUE; END_IF;
END_PROGRAM
```

### Program Logical/BagMachine_Section/FP/Axis2/A2_Cycle (IEC) - A new program
